// TwinCAT 3 PLC project Main
// ProgramVersion: 3.1.4023.0
// libraries:
//   Tc2_Standard, * (Beckhoff Automation GmbH)
//   Tc2_System, * (Beckhoff Automation GmbH)
//   Tc3_Module, * (Beckhoff Automation GmbH)
//   TcUnit, * (www.tcunit.org)
//   mobject-constants-datatype-limits,1.0.0,mobject
//   mobject-converters,1.0.2,mobject
// project tree:
//   / PlcTask.TcTTO
//   POUs/ MAIN.TcPOU
//   Tests/ BOOL_TO_TestSuite.TcPOU, BYTE_TO_TestSuite.TcPOU, DATE_TO_TestSuite.TcPOU, DINT_TO_TestSuite.TcPOU, DT_TO_TestSuite.TcPOU, DWORD_TO_TestSuite.TcPOU, INT_TO_TestSuite.TcPOU, LINT_TO_TestSuite.TcPOU, LREAL_TO_TestSuite.TcPOU, LWORD_TO_TestSuite.TcPOU, REAL_TO_TestSuite.TcPOU, SINT_TO_TestSuite.TcPOU, STRING_TO_TestSuite.TcPOU, TIME_TO_TestSuite.TcPOU, TOD_TO_TestSuite.TcPOU, UDINT_TO_TestSuite.TcPOU, UINT_TO_TestSuite.TcPOU, ULINT_TO_TestSuite.TcPOU, USINT_TO_TestSuite.TcPOU, WORD_TO_TestSuite.TcPOU
// real-time tasks:
//   TASK PlcTask: cycle T#10ms, priority 20, ADS port 350

CONFIGURATION Main
    RESOURCE PLC ON TwinCAT3
        TASK PlcTask(INTERVAL := T#10ms, PRIORITY := 20);
        PROGRAM MAIN WITH PlcTask : MAIN;
    END_RESOURCE
END_CONFIGURATION

// ---- POUs/MAIN.TcPOU
PROGRAM MAIN
VAR
	BOOL_TO_TestSuite : BOOL_TO_TestSuite;
	BYTE_TO_TestSuite : BYTE_TO_TestSuite;
	WORD_TO_TestSuite : WORD_TO_TestSuite;
	DWORD_TO_TestSuite : DWORD_TO_TestSuite;
	LWORD_TO_TestSuite : LWORD_TO_TestSuite;
	SINT_TO_TestSuite : SINT_TO_TestSuite;
	INT_TO_TestSuite : INT_TO_TestSuite;
	DINT_TO_TestSuite : DINT_TO_TestSuite;
	LINT_TO_TestSuite : LINT_TO_TestSuite;
	USINT_TO_TestSuite : USINT_TO_TestSuite;
	UINT_TO_TestSuite : UINT_TO_TestSuite;
	UDINT_TO_TestSuite : UDINT_TO_TestSuite;
	ULINT_TO_TestSuite : ULINT_TO_TestSuite;
	REAL_TO_TestSuite : REAL_TO_TestSuite;
	LREAL_TO_TestSuite : LREAL_TO_TestSuite;
	TIME_TO_TestSuite : TIME_TO_TestSuite;
	TOD_TO_TestSuite : TOD_TO_TestSuite;
	DATE_TO_TestSuite : DATE_TO_TestSuite;
	DT_TO_TestSuite : DT_TO_TestSuite;
	STRING_TO_TestSuite : STRING_TO_TestSuite;
END_VAR

TcUnit.RUN();

END_PROGRAM

// ---- Tests/BOOL_TO_TestSuite.TcPOU
FUNCTION_BLOCK PUBLIC BOOL_TO_TestSuite EXTENDS TcUnit.FB_TestSuite
VAR
END_VAR

Check_BOOL_TO_BOOL_Max();
Check_BOOL_TO_BOOL_Min();
Check_BOOL_TO_BYTE_Max();
Check_BOOL_TO_BYTE_Min();
Check_BOOL_TO_WORD_Max();
Check_BOOL_TO_WORD_Min();
Check_BOOL_TO_DWORD_Max();
Check_BOOL_TO_DWORD_Min();
Check_BOOL_TO_LWORD_Max();
Check_BOOL_TO_LWORD_Min();
Check_BOOL_TO_SINT_Max();
Check_BOOL_TO_SINT_Min();
Check_BOOL_TO_INT_Max();
Check_BOOL_TO_INT_Min();
Check_BOOL_TO_DINT_Max();
Check_BOOL_TO_DINT_Min();
Check_BOOL_TO_LINT_Max();
Check_BOOL_TO_LINT_Min();
Check_BOOL_TO_USINT_Max();
Check_BOOL_TO_USINT_Min();
Check_BOOL_TO_UINT_Max();
Check_BOOL_TO_UINT_Min();
Check_BOOL_TO_UDINT_Max();
Check_BOOL_TO_UDINT_Min();
Check_BOOL_TO_ULINT_Max();
Check_BOOL_TO_ULINT_Min();
Check_BOOL_TO_REAL_Max();
Check_BOOL_TO_REAL_Min();
Check_BOOL_TO_LREAL_Max();
Check_BOOL_TO_LREAL_Min();
Check_BOOL_TO_TIME_Max();
Check_BOOL_TO_TIME_Min();
Check_BOOL_TO_TOD_Max();
Check_BOOL_TO_TOD_Min();
Check_BOOL_TO_DATE_Max();
Check_BOOL_TO_DATE_Min();
Check_BOOL_TO_DT_Max();
Check_BOOL_TO_DT_Min();
Check_BOOL_TO_STRING_Max();
Check_BOOL_TO_STRING_Min();

METHOD PUBLIC Check_BOOL_TO_BOOL_Min
VAR
	value : BOOL := DatatypeLimits.BOOL_MIN_VALUE;
	actual : BOOL;
	converted : BOOL;
	equal : BOOL;
END_VAR
TEST('Check_BOOL_TO_BOOL_Min');

// @TEST-RUN
converted := TryConvert_BOOL_TO_Destination(value, actual);
equal := actual = value;

// @TEST-ASSERT
AssertTrue(Condition := equal, Message := 'Did not convert BOOL to BOOL correctly');
AssertTrue(Condition := converted, Message := 'Did not report BOOL to BOOL conversion was successful');

TEST_FINISHED();
END_METHOD

METHOD PUBLIC Check_BOOL_TO_BOOL_Max
VAR
	value : BOOL := DatatypeLimits.BOOL_MAX_VALUE;
	actual : BOOL;
	converted : BOOL;
	equal : BOOL;
END_VAR
TEST('Check_BOOL_TO_BOOL_Max');

// @TEST-RUN
converted := TryConvert_BOOL_TO_Destination(value, actual);
equal := actual = value;

// @TEST-ASSERT
AssertTrue(Condition := equal, Message := 'Did not convert BOOL to BOOL correctly');
AssertTrue(Condition := converted, Message := 'Did not report BOOL to BOOL conversion was successful');

TEST_FINISHED();
END_METHOD

METHOD PUBLIC Check_BOOL_TO_BYTE_Min
VAR
	value : BOOL := DatatypeLimits.BOOL_MIN_VALUE;
	actual : BYTE;
	converted : BOOL;
	equal : BOOL;
END_VAR
TEST('Check_BOOL_TO_BYTE_Min');

// @TEST-RUN
converted := TryConvert_BOOL_TO_Destination(value, actual);
equal := actual = BOOL_TO_BYTE(value);

// @TEST-ASSERT
AssertTrue(Condition := equal, Message := 'Did not convert BOOL to BYTE correctly');
AssertTrue(Condition := converted, Message := 'Did not report BOOL to BYTE conversion was successful');

TEST_FINISHED();
END_METHOD

METHOD PUBLIC Check_BOOL_TO_BYTE_Max
VAR
	value : BOOL := DatatypeLimits.BOOL_MAX_VALUE;
	actual : BYTE;
	converted : BOOL;
	equal : BOOL;
END_VAR
TEST('Check_BOOL_TO_BYTE_Max');

// @TEST-RUN
converted := TryConvert_BOOL_TO_Destination(value, actual);
equal := actual = BOOL_TO_BYTE(value);

// @TEST-ASSERT
AssertTrue(Condition := equal, Message := 'Did not convert BOOL to BYTE correctly');
AssertTrue(Condition := converted, Message := 'Did not report BOOL to BYTE conversion was successful');

TEST_FINISHED();
END_METHOD

METHOD PUBLIC Check_BOOL_TO_DATE_Min
VAR
	value : BOOL := DatatypeLimits.BOOL_MIN_VALUE;
	actual : DATE;
	converted : BOOL;
	equal : BOOL;
END_VAR
TEST('Check_BOOL_TO_DATE_Min');

// @TEST-RUN
converted := TryConvert_BOOL_TO_Destination(value, actual);
equal := actual = BOOL_TO_DATE(value);

// @TEST-ASSERT
AssertTrue(Condition := equal, Message := 'Did not convert BOOL to DATE correctly');
AssertTrue(Condition := converted, Message := 'Did not report BOOL to DATE conversion was successful');

TEST_FINISHED();
END_METHOD

METHOD PUBLIC Check_BOOL_TO_DATE_Max
VAR
	value : BOOL := DatatypeLimits.BOOL_MAX_VALUE;
	actual : DATE;
	converted : BOOL;
	equal : BOOL;
END_VAR
TEST('Check_BOOL_TO_DATE_Max');

// @TEST-RUN
converted := TryConvert_BOOL_TO_Destination(value, actual);
equal := actual = BOOL_TO_DATE(value);

// @TEST-ASSERT
AssertTrue(Condition := equal, Message := 'Did not convert BOOL to DATE correctly');
AssertTrue(Condition := converted, Message := 'Did not report BOOL to DATE conversion was successful');

TEST_FINISHED();
END_METHOD

METHOD PUBLIC Check_BOOL_TO_DINT_Min
VAR
	value : BOOL := DatatypeLimits.BOOL_MIN_VALUE;
	actual : DINT;
	converted : BOOL;
	equal : BOOL;
END_VAR
TEST('Check_BOOL_TO_DINT_Min');

// @TEST-RUN
converted := TryConvert_BOOL_TO_Destination(value, actual);
equal := actual = BOOL_TO_DINT(value);

// @TEST-ASSERT
AssertTrue(Condition := equal, Message := 'Did not convert BOOL to DINT correctly');
AssertTrue(Condition := converted, Message := 'Did not report BOOL to DINT conversion was successful');

TEST_FINISHED();
END_METHOD

METHOD PUBLIC Check_BOOL_TO_DINT_Max
VAR
	value : BOOL := DatatypeLimits.BOOL_MAX_VALUE;
	actual : DINT;
	converted : BOOL;
	equal : BOOL;
END_VAR
TEST('Check_BOOL_TO_DINT_Max');

// @TEST-RUN
converted := TryConvert_BOOL_TO_Destination(value, actual);
equal := actual = BOOL_TO_DINT(value);

// @TEST-ASSERT
AssertTrue(Condition := equal, Message := 'Did not convert BOOL to DINT correctly');
AssertTrue(Condition := converted, Message := 'Did not report BOOL to DINT conversion was successful');

TEST_FINISHED();
END_METHOD

METHOD PUBLIC Check_BOOL_TO_DT_Min
VAR
	value : BOOL := DatatypeLimits.BOOL_MIN_VALUE;
	actual : DT;
	converted : BOOL;
	equal : BOOL;
END_VAR
TEST('Check_BOOL_TO_DT_Min');

// @TEST-RUN
converted := TryConvert_BOOL_TO_Destination(value, actual);
equal := actual = BOOL_TO_DT(value);

// @TEST-ASSERT
AssertTrue(Condition := equal, Message := 'Did not convert BOOL to DT correctly');
AssertTrue(Condition := converted, Message := 'Did not report BOOL to DT conversion was successful');

TEST_FINISHED();
END_METHOD

METHOD PUBLIC Check_BOOL_TO_DT_Max
VAR
	value : BOOL := DatatypeLimits.BOOL_MAX_VALUE;
	actual : DT;
	converted : BOOL;
	equal : BOOL;
END_VAR
TEST('Check_BOOL_TO_DT_Max');

// @TEST-RUN
converted := TryConvert_BOOL_TO_Destination(value, actual);
equal := actual = BOOL_TO_DT(value);

// @TEST-ASSERT
AssertTrue(Condition := equal, Message := 'Did not convert BOOL to DT correctly');
AssertTrue(Condition := converted, Message := 'Did not report BOOL to DT conversion was successful');

TEST_FINISHED();
END_METHOD

METHOD PUBLIC Check_BOOL_TO_DWORD_Min
VAR
	value : BOOL := DatatypeLimits.BOOL_MIN_VALUE;
	actual : DWORD;
	converted : BOOL;
	equal : BOOL;
END_VAR
TEST('Check_BOOL_TO_DWORD_Min');

// @TEST-RUN
converted := TryConvert_BOOL_TO_Destination(value, actual);
equal := actual = BOOL_TO_DWORD(value);

// @TEST-ASSERT
AssertTrue(Condition := equal, Message := 'Did not convert BOOL to DWORD correctly');
AssertTrue(Condition := converted, Message := 'Did not report BOOL to DWORD conversion was successful');

TEST_FINISHED();
END_METHOD

METHOD PUBLIC Check_BOOL_TO_DWORD_Max
VAR
	value : BOOL := DatatypeLimits.BOOL_MAX_VALUE;
	actual : DWORD;
	converted : BOOL;
	equal : BOOL;
END_VAR
TEST('Check_BOOL_TO_DWORD_Max');

// @TEST-RUN
converted := TryConvert_BOOL_TO_Destination(value, actual);
equal := actual = BOOL_TO_DWORD(value);

// @TEST-ASSERT
AssertTrue(Condition := equal, Message := 'Did not convert BOOL to DWORD correctly');
AssertTrue(Condition := converted, Message := 'Did not report BOOL to DWORD conversion was successful');

TEST_FINISHED();
END_METHOD

METHOD PUBLIC Check_BOOL_TO_INT_Min
VAR
	value : BOOL := DatatypeLimits.BOOL_MIN_VALUE;
	actual : INT;
	converted : BOOL;
	equal : BOOL;
END_VAR
TEST('Check_BOOL_TO_INT_Min');

// @TEST-RUN
converted := TryConvert_BOOL_TO_Destination(value, actual);
equal := actual = BOOL_TO_INT(value);

// @TEST-ASSERT
AssertTrue(Condition := equal, Message := 'Did not convert BOOL to INT correctly');
AssertTrue(Condition := converted, Message := 'Did not report BOOL to INT conversion was successful');

TEST_FINISHED();
END_METHOD

METHOD PUBLIC Check_BOOL_TO_INT_Max
VAR
	value : BOOL := DatatypeLimits.BOOL_MAX_VALUE;
	actual : INT;
	converted : BOOL;
	equal : BOOL;
END_VAR
TEST('Check_BOOL_TO_INT_Max');

// @TEST-RUN
converted := TryConvert_BOOL_TO_Destination(value, actual);
equal := actual = BOOL_TO_INT(value);

// @TEST-ASSERT
AssertTrue(Condition := equal, Message := 'Did not convert BOOL to INT correctly');
AssertTrue(Condition := converted, Message := 'Did not report BOOL to INT conversion was successful');

TEST_FINISHED();
END_METHOD

METHOD PUBLIC Check_BOOL_TO_LINT_Min
VAR
	value : BOOL := DatatypeLimits.BOOL_MIN_VALUE;
	actual : LINT;
	converted : BOOL;
	equal : BOOL;
END_VAR
TEST('Check_BOOL_TO_LINT_Min');

// @TEST-RUN
converted := TryConvert_BOOL_TO_Destination(value, actual);
equal := actual = BOOL_TO_LINT(value);

// @TEST-ASSERT
AssertTrue(Condition := equal, Message := 'Did not convert BOOL to LINT correctly');
AssertTrue(Condition := converted, Message := 'Did not report BOOL to LINT conversion was successful');

TEST_FINISHED();
END_METHOD

METHOD PUBLIC Check_BOOL_TO_LINT_Max
VAR
	value : BOOL := DatatypeLimits.BOOL_MAX_VALUE;
	actual : LINT;
	converted : BOOL;
	equal : BOOL;
END_VAR
TEST('Check_BOOL_TO_LINT_Max');

// @TEST-RUN
converted := TryConvert_BOOL_TO_Destination(value, actual);
equal := actual = BOOL_TO_LINT(value);

// @TEST-ASSERT
AssertTrue(Condition := equal, Message := 'Did not convert BOOL to LINT correctly');
AssertTrue(Condition := converted, Message := 'Did not report BOOL to LINT conversion was successful');

TEST_FINISHED();
END_METHOD

METHOD PUBLIC Check_BOOL_TO_LREAL_Min
VAR
	value : BOOL := DatatypeLimits.BOOL_MIN_VALUE;
	actual : LREAL;
	converted : BOOL;
	equal : BOOL;
END_VAR
TEST('Check_BOOL_TO_LREAL_Min');

// @TEST-RUN
converted := TryConvert_BOOL_TO_Destination(value, actual);
equal := actual = BOOL_TO_LREAL(value);

// @TEST-ASSERT
AssertTrue(Condition := equal, Message := 'Did not convert BOOL to LREAL correctly');
AssertTrue(Condition := converted, Message := 'Did not report BOOL to LREAL conversion was successful');

TEST_FINISHED();
END_METHOD

METHOD PUBLIC Check_BOOL_TO_LREAL_Max
VAR
	value : BOOL := DatatypeLimits.BOOL_MAX_VALUE;
	actual : LREAL;
	converted : BOOL;
	equal : BOOL;
END_VAR
TEST('Check_BOOL_TO_LREAL_Max');

// @TEST-RUN
converted := TryConvert_BOOL_TO_Destination(value, actual);
equal := actual = BOOL_TO_LREAL(value);

// @TEST-ASSERT
AssertTrue(Condition := equal, Message := 'Did not convert BOOL to LREAL correctly');
AssertTrue(Condition := converted, Message := 'Did not report BOOL to LREAL conversion was successful');

TEST_FINISHED();
END_METHOD

METHOD PUBLIC Check_BOOL_TO_LWORD_Min
VAR
	value : BOOL := DatatypeLimits.BOOL_MIN_VALUE;
	actual : LWORD;
	converted : BOOL;
	equal : BOOL;
END_VAR
TEST('Check_BOOL_TO_LWORD_Min');

// @TEST-RUN
converted := TryConvert_BOOL_TO_Destination(value, actual);
equal := actual = BOOL_TO_LWORD(value);

// @TEST-ASSERT
AssertTrue(Condition := equal, Message := 'Did not convert BOOL to LWORD correctly');
AssertTrue(Condition := converted, Message := 'Did not report BOOL to LWORD conversion was successful');

TEST_FINISHED();
END_METHOD

METHOD PUBLIC Check_BOOL_TO_LWORD_Max
VAR
	value : BOOL := DatatypeLimits.BOOL_MAX_VALUE;
	actual : LWORD;
	converted : BOOL;
	equal : BOOL;
END_VAR
TEST('Check_BOOL_TO_LWORD_Max');

// @TEST-RUN
converted := TryConvert_BOOL_TO_Destination(value, actual);
equal := actual = BOOL_TO_LWORD(value);

// @TEST-ASSERT
AssertTrue(Condition := equal, Message := 'Did not convert BOOL to LWORD correctly');
AssertTrue(Condition := converted, Message := 'Did not report BOOL to LWORD conversion was successful');

TEST_FINISHED();
END_METHOD

METHOD PUBLIC Check_BOOL_TO_REAL_Min
VAR
	value : BOOL := DatatypeLimits.BOOL_MIN_VALUE;
	actual : REAL;
	converted : BOOL;
	equal : BOOL;
END_VAR
TEST('Check_BOOL_TO_REAL_Min');

// @TEST-RUN
converted := TryConvert_BOOL_TO_Destination(value, actual);
equal := actual = BOOL_TO_REAL(value);

// @TEST-ASSERT
AssertTrue(Condition := equal, Message := 'Did not convert BOOL to REAL correctly');
AssertTrue(Condition := converted, Message := 'Did not report BOOL to REAL conversion was successful');

TEST_FINISHED();
END_METHOD

METHOD PUBLIC Check_BOOL_TO_REAL_Max
VAR
	value : BOOL := DatatypeLimits.BOOL_MAX_VALUE;
	actual : REAL;
	converted : BOOL;
	equal : BOOL;
END_VAR
TEST('Check_BOOL_TO_REAL_Max');

// @TEST-RUN
converted := TryConvert_BOOL_TO_Destination(value, actual);
equal := actual = BOOL_TO_REAL(value);

// @TEST-ASSERT
AssertTrue(Condition := equal, Message := 'Did not convert BOOL to REAL correctly');
AssertTrue(Condition := converted, Message := 'Did not report BOOL to REAL conversion was successful');

TEST_FINISHED();
END_METHOD

METHOD PUBLIC Check_BOOL_TO_SINT_Min
VAR
	value : BOOL := DatatypeLimits.BOOL_MIN_VALUE;
	actual : SINT;
	converted : BOOL;
	equal : BOOL;
END_VAR
TEST('Check_BOOL_TO_SINT_Min');

// @TEST-RUN
converted := TryConvert_BOOL_TO_Destination(value, actual);
equal := actual = BOOL_TO_SINT(value);

// @TEST-ASSERT
AssertTrue(Condition := equal, Message := 'Did not convert BOOL to SINT correctly');
AssertTrue(Condition := converted, Message := 'Did not report BOOL to SINT conversion was successful');

TEST_FINISHED();
END_METHOD

METHOD PUBLIC Check_BOOL_TO_SINT_Max
VAR
	value : BOOL := DatatypeLimits.BOOL_MAX_VALUE;
	actual : SINT;
	converted : BOOL;
	equal : BOOL;
END_VAR
TEST('Check_BOOL_TO_SINT_Max');

// @TEST-RUN
converted := TryConvert_BOOL_TO_Destination(value, actual);
equal := actual = BOOL_TO_SINT(value);

// @TEST-ASSERT
AssertTrue(Condition := equal, Message := 'Did not convert BOOL to SINT correctly');
AssertTrue(Condition := converted, Message := 'Did not report BOOL to SINT conversion was successful');

TEST_FINISHED();
END_METHOD

METHOD PUBLIC Check_BOOL_TO_STRING_Min
VAR
	value : BOOL := DatatypeLimits.BOOL_MIN_VALUE;
	actual : STRING;
	converted : BOOL;
	equal : BOOL;
END_VAR
TEST('Check_BOOL_TO_STRING_Min');

// @TEST-RUN
converted := TryConvert_BOOL_TO_Destination(value, actual);
equal := actual = BOOL_TO_STRING(value);

// @TEST-ASSERT
AssertTrue(Condition := equal, Message := 'Did not convert BOOL to STRING correctly');
AssertTrue(Condition := converted, Message := 'Did not report BOOL to STRING conversion was successful');

TEST_FINISHED();
END_METHOD

METHOD PUBLIC Check_BOOL_TO_STRING_Max
VAR
	value : BOOL := DatatypeLimits.BOOL_MAX_VALUE;
	actual : STRING;
	converted : BOOL;
	equal : BOOL;
END_VAR
TEST('Check_BOOL_TO_STRING_Max');

// @TEST-RUN
converted := TryConvert_BOOL_TO_Destination(value, actual);
equal := actual = BOOL_TO_STRING(value);

// @TEST-ASSERT
AssertTrue(Condition := equal, Message := 'Did not convert BOOL to STRING correctly');
AssertTrue(Condition := converted, Message := 'Did not report BOOL to STRING conversion was successful');

TEST_FINISHED();
END_METHOD

METHOD PUBLIC Check_BOOL_TO_TIME_Min
VAR
	value : BOOL := DatatypeLimits.BOOL_MIN_VALUE;
	actual : TIME;
	converted : BOOL;
	equal : BOOL;
END_VAR
TEST('Check_BOOL_TO_TIME_Min');

// @TEST-RUN
converted := TryConvert_BOOL_TO_Destination(value, actual);
equal := actual = BOOL_TO_TIME(value);

// @TEST-ASSERT
AssertTrue(Condition := equal, Message := 'Did not convert BOOL to TIME correctly');
AssertTrue(Condition := converted, Message := 'Did not report BOOL to TIME conversion was successful');

TEST_FINISHED();
END_METHOD

METHOD PUBLIC Check_BOOL_TO_TIME_Max
VAR
	value : BOOL := DatatypeLimits.BOOL_MAX_VALUE;
	actual : TIME;
	converted : BOOL;
	equal : BOOL;
END_VAR
TEST('Check_BOOL_TO_TIME_Max');

// @TEST-RUN
converted := TryConvert_BOOL_TO_Destination(value, actual);
equal := actual = BOOL_TO_TIME(value);

// @TEST-ASSERT
AssertTrue(Condition := equal, Message := 'Did not convert BOOL to TIME correctly');
AssertTrue(Condition := converted, Message := 'Did not report BOOL to TIME conversion was successful');

TEST_FINISHED();
END_METHOD

METHOD PUBLIC Check_BOOL_TO_TOD_Min
VAR
	value : BOOL := DatatypeLimits.BOOL_MIN_VALUE;
	actual : TOD;
	converted : BOOL;
	equal : BOOL;
END_VAR
TEST('Check_BOOL_TO_TOD_Min');

// @TEST-RUN
converted := TryConvert_BOOL_TO_Destination(value, actual);
equal := actual = BOOL_TO_TOD(value);

// @TEST-ASSERT
AssertTrue(Condition := equal, Message := 'Did not convert BOOL to TOD correctly');
AssertTrue(Condition := converted, Message := 'Did not report BOOL to TOD conversion was successful');

TEST_FINISHED();
END_METHOD

METHOD PUBLIC Check_BOOL_TO_TOD_Max
VAR
	value : BOOL := DatatypeLimits.BOOL_MAX_VALUE;
	actual : TOD;
	converted : BOOL;
	equal : BOOL;
END_VAR
TEST('Check_BOOL_TO_TOD_Max');

// @TEST-RUN
converted := TryConvert_BOOL_TO_Destination(value, actual);
equal := actual = BOOL_TO_TOD(value);

// @TEST-ASSERT
AssertTrue(Condition := equal, Message := 'Did not convert BOOL to TOD correctly');
AssertTrue(Condition := converted, Message := 'Did not report BOOL to TOD conversion was successful');

TEST_FINISHED();
END_METHOD

METHOD PUBLIC Check_BOOL_TO_UDINT_Min
VAR
	value : BOOL := DatatypeLimits.BOOL_MIN_VALUE;
	actual : UDINT;
	converted : BOOL;
	equal : BOOL;
END_VAR
TEST('Check_BOOL_TO_UDINT_Min');

// @TEST-RUN
converted := TryConvert_BOOL_TO_Destination(value, actual);
equal := actual = BOOL_TO_UDINT(value);

// @TEST-ASSERT
AssertTrue(Condition := equal, Message := 'Did not convert BOOL to UDINT correctly');
AssertTrue(Condition := converted, Message := 'Did not report BOOL to UDINT conversion was successful');

TEST_FINISHED();
END_METHOD

METHOD PUBLIC Check_BOOL_TO_UDINT_Max
VAR
	value : BOOL := DatatypeLimits.BOOL_MAX_VALUE;
	actual : UDINT;
	converted : BOOL;
	equal : BOOL;
END_VAR
TEST('Check_BOOL_TO_UDINT_Max');

// @TEST-RUN
converted := TryConvert_BOOL_TO_Destination(value, actual);
equal := actual = BOOL_TO_UDINT(value);

// @TEST-ASSERT
AssertTrue(Condition := equal, Message := 'Did not convert BOOL to UDINT correctly');
AssertTrue(Condition := converted, Message := 'Did not report BOOL to UDINT conversion was successful');

TEST_FINISHED();
END_METHOD

METHOD PUBLIC Check_BOOL_TO_UINT_Min
VAR
	value : BOOL := DatatypeLimits.BOOL_MIN_VALUE;
	actual : UINT;
	converted : BOOL;
	equal : BOOL;
END_VAR
TEST('Check_BOOL_TO_UINT_Min');

// @TEST-RUN
converted := TryConvert_BOOL_TO_Destination(value, actual);
equal := actual = BOOL_TO_UINT(value);

// @TEST-ASSERT
AssertTrue(Condition := equal, Message := 'Did not convert BOOL to UINT correctly');
AssertTrue(Condition := converted, Message := 'Did not report BOOL to UINT conversion was successful');

TEST_FINISHED();
END_METHOD

METHOD PUBLIC Check_BOOL_TO_UINT_Max
VAR
	value : BOOL := DatatypeLimits.BOOL_MAX_VALUE;
	actual : UINT;
	converted : BOOL;
	equal : BOOL;
END_VAR
TEST('Check_BOOL_TO_UINT_Max');

// @TEST-RUN
converted := TryConvert_BOOL_TO_Destination(value, actual);
equal := actual = BOOL_TO_UINT(value);

// @TEST-ASSERT
AssertTrue(Condition := equal, Message := 'Did not convert BOOL to UINT correctly');
AssertTrue(Condition := converted, Message := 'Did not report BOOL to UINT conversion was successful');

TEST_FINISHED();
END_METHOD

METHOD PUBLIC Check_BOOL_TO_ULINT_Min
VAR
	value : BOOL := DatatypeLimits.BOOL_MIN_VALUE;
	actual : ULINT;
	converted : BOOL;
	equal : BOOL;
END_VAR
TEST('Check_BOOL_TO_ULINT_Min');

// @TEST-RUN
converted := TryConvert_BOOL_TO_Destination(value, actual);
equal := actual = BOOL_TO_ULINT(value);

// @TEST-ASSERT
AssertTrue(Condition := equal, Message := 'Did not convert BOOL to ULINT correctly');
AssertTrue(Condition := converted, Message := 'Did not report BOOL to ULINT conversion was successful');

TEST_FINISHED();
END_METHOD

METHOD PUBLIC Check_BOOL_TO_ULINT_Max
VAR
	value : BOOL := DatatypeLimits.BOOL_MAX_VALUE;
	actual : ULINT;
	converted : BOOL;
	equal : BOOL;
END_VAR
TEST('Check_BOOL_TO_ULINT_Max');

// @TEST-RUN
converted := TryConvert_BOOL_TO_Destination(value, actual);
equal := actual = BOOL_TO_ULINT(value);

// @TEST-ASSERT
AssertTrue(Condition := equal, Message := 'Did not convert BOOL to ULINT correctly');
AssertTrue(Condition := converted, Message := 'Did not report BOOL to ULINT conversion was successful');

TEST_FINISHED();
END_METHOD

METHOD PUBLIC Check_BOOL_TO_USINT_Min
VAR
	value : BOOL := DatatypeLimits.BOOL_MIN_VALUE;
	actual : USINT;
	converted : BOOL;
	equal : BOOL;
END_VAR
TEST('Check_BOOL_TO_USINT_Min');

// @TEST-RUN
converted := TryConvert_BOOL_TO_Destination(value, actual);
equal := actual = BOOL_TO_USINT(value);

// @TEST-ASSERT
AssertTrue(Condition := equal, Message := 'Did not convert BOOL to USINT correctly');
AssertTrue(Condition := converted, Message := 'Did not report BOOL to USINT conversion was successful');

TEST_FINISHED();
END_METHOD

METHOD PUBLIC Check_BOOL_TO_USINT_Max
VAR
	value : BOOL := DatatypeLimits.BOOL_MAX_VALUE;
	actual : USINT;
	converted : BOOL;
	equal : BOOL;
END_VAR
TEST('Check_BOOL_TO_USINT_Max');

// @TEST-RUN
converted := TryConvert_BOOL_TO_Destination(value, actual);
equal := actual = BOOL_TO_USINT(value);

// @TEST-ASSERT
AssertTrue(Condition := equal, Message := 'Did not convert BOOL to USINT correctly');
AssertTrue(Condition := converted, Message := 'Did not report BOOL to USINT conversion was successful');

TEST_FINISHED();
END_METHOD

METHOD PUBLIC Check_BOOL_TO_WORD_Min
VAR
	value : BOOL := DatatypeLimits.BOOL_MIN_VALUE;
	actual : WORD;
	converted : BOOL;
	equal : BOOL;
END_VAR
TEST('Check_BOOL_TO_WORD_Min');

// @TEST-RUN
converted := TryConvert_BOOL_TO_Destination(value, actual);
equal := actual = BOOL_TO_WORD(value);

// @TEST-ASSERT
AssertTrue(Condition := equal, Message := 'Did not convert BOOL to WORD correctly');
AssertTrue(Condition := converted, Message := 'Did not report BOOL to WORD conversion was successful');

TEST_FINISHED();
END_METHOD

METHOD PUBLIC Check_BOOL_TO_WORD_Max
VAR
	value : BOOL := DatatypeLimits.BOOL_MAX_VALUE;
	actual : WORD;
	converted : BOOL;
	equal : BOOL;
END_VAR
TEST('Check_BOOL_TO_WORD_Max');

// @TEST-RUN
converted := TryConvert_BOOL_TO_Destination(value, actual);
equal := actual = BOOL_TO_WORD(value);

// @TEST-ASSERT
AssertTrue(Condition := equal, Message := 'Did not convert BOOL to WORD correctly');
AssertTrue(Condition := converted, Message := 'Did not report BOOL to WORD conversion was successful');

TEST_FINISHED();
END_METHOD

END_FUNCTION_BLOCK

// ---- Tests/BYTE_TO_TestSuite.TcPOU
FUNCTION_BLOCK PUBLIC BYTE_TO_TestSuite EXTENDS TcUnit.FB_TestSuite
VAR
END_VAR

Check_BYTE_TO_BOOL_Max();
Check_BYTE_TO_BOOL_Min();
Check_BYTE_TO_BYTE_Max();
Check_BYTE_TO_BYTE_Min();
Check_BYTE_TO_WORD_Max();
Check_BYTE_TO_WORD_Min();
Check_BYTE_TO_DWORD_Max();
Check_BYTE_TO_DWORD_Min();
Check_BYTE_TO_LWORD_Max();
Check_BYTE_TO_LWORD_Min();
Check_BYTE_TO_SINT_Max();
Check_BYTE_TO_SINT_Min();
Check_BYTE_TO_SINT_TooHigh();
Check_BYTE_TO_INT_Max();
Check_BYTE_TO_INT_Min();
Check_BYTE_TO_DINT_Max();
Check_BYTE_TO_DINT_Min();
Check_BYTE_TO_LINT_Max();
Check_BYTE_TO_LINT_Min();
Check_BYTE_TO_USINT_Max();
Check_BYTE_TO_USINT_Min();
Check_BYTE_TO_UINT_Max();
Check_BYTE_TO_UINT_Min();
Check_BYTE_TO_UDINT_Max();
Check_BYTE_TO_UDINT_Min();
Check_BYTE_TO_ULINT_Max();
Check_BYTE_TO_ULINT_Min();
Check_BYTE_TO_REAL_Max();
Check_BYTE_TO_REAL_Min();
Check_BYTE_TO_LREAL_Max();
Check_BYTE_TO_LREAL_Min();
Check_BYTE_TO_TIME_Max();
Check_BYTE_TO_TIME_Min();
Check_BYTE_TO_TOD_Max();
Check_BYTE_TO_TOD_Min();
Check_BYTE_TO_DATE_Max();
Check_BYTE_TO_DATE_Min();
Check_BYTE_TO_DT_Max();
Check_BYTE_TO_DT_Min();
Check_BYTE_TO_STRING_Max();
Check_BYTE_TO_STRING_Min();

METHOD PUBLIC Check_BYTE_TO_BOOL_Min
VAR
	value : BYTE := DatatypeLimits.BYTE_MIN_VALUE;
	actual : BOOL;
	converted : BOOL;
	equal : BOOL;
END_VAR
TEST('Check_BYTE_TO_BOOL_Min');

// @TEST-RUN
converted := TryConvert_BYTE_TO_Destination(value, actual);
equal := actual = BYTE_TO_BOOL(value);

// @TEST-ASSERT
AssertTrue(Condition := equal, Message := 'Did not convert BYTE to BOOL correctly');
AssertTrue(Condition := converted, Message := 'Did not report BYTE to BOOL conversion was successful');

TEST_FINISHED();
END_METHOD

METHOD PUBLIC Check_BYTE_TO_BOOL_Max
VAR
	value : BYTE := DatatypeLimits.BYTE_MAX_VALUE;
	actual : BOOL;
	converted : BOOL;
	equal : BOOL;
END_VAR
TEST('Check_BYTE_TO_BOOL_Max');

// @TEST-RUN
converted := TryConvert_BYTE_TO_Destination(value, actual);
equal := actual = BYTE_TO_BOOL(value);

// @TEST-ASSERT
AssertTrue(Condition := equal, Message := 'Did not convert BYTE to BOOL correctly');
AssertTrue(Condition := converted, Message := 'Did not report BYTE to BOOL conversion was successful');

TEST_FINISHED();
END_METHOD

METHOD PUBLIC Check_BYTE_TO_BYTE_Min
VAR
	value : BYTE := DatatypeLimits.BYTE_MIN_VALUE;
	actual : BYTE;
	converted : BOOL;
	equal : BOOL;
END_VAR
TEST('Check_BYTE_TO_BYTE_Min');

// @TEST-RUN
converted := TryConvert_BYTE_TO_Destination(value, actual);
equal := actual = value;

// @TEST-ASSERT
AssertTrue(Condition := equal, Message := 'Did not convert BYTE to BYTE correctly');
AssertTrue(Condition := converted, Message := 'Did not report BYTE to BYTE conversion was successful');

TEST_FINISHED();
END_METHOD

METHOD PUBLIC Check_BYTE_TO_BYTE_Max
VAR
	value : BYTE := DatatypeLimits.BYTE_MAX_VALUE;
	actual : BYTE;
	converted : BOOL;
	equal : BOOL;
END_VAR
TEST('Check_BYTE_TO_BYTE_Max');

// @TEST-RUN
converted := TryConvert_BYTE_TO_Destination(value, actual);
equal := actual = value;

// @TEST-ASSERT
AssertTrue(Condition := equal, Message := 'Did not convert BYTE to BYTE correctly');
AssertTrue(Condition := converted, Message := 'Did not report BYTE to BYTE conversion was successful');

TEST_FINISHED();
END_METHOD

METHOD PUBLIC Check_BYTE_TO_DATE_Min
VAR
	value : BYTE := DatatypeLimits.BYTE_MIN_VALUE;
	actual : DATE;
	converted : BOOL;
	equal : BOOL;
END_VAR
TEST('Check_BYTE_TO_DATE_Min');

// @TEST-RUN
converted := TryConvert_BYTE_TO_Destination(value, actual);
equal := actual = BYTE_TO_DATE(value);

// @TEST-ASSERT
AssertTrue(Condition := equal, Message := 'Did not convert BYTE to DATE correctly');
AssertTrue(Condition := converted, Message := 'Did not report BYTE to DATE conversion was successful');

TEST_FINISHED();
END_METHOD

METHOD PUBLIC Check_BYTE_TO_DATE_Max
VAR
	value : BYTE := DatatypeLimits.BYTE_MAX_VALUE;
	actual : DATE;
	converted : BOOL;
	equal : BOOL;
END_VAR
TEST('Check_BYTE_TO_DATE_Max');

// @TEST-RUN
converted := TryConvert_BYTE_TO_Destination(value, actual);
equal := actual = BYTE_TO_DATE(value);

// @TEST-ASSERT
AssertTrue(Condition := equal, Message := 'Did not convert BYTE to DATE correctly');
AssertTrue(Condition := converted, Message := 'Did not report BYTE to DATE conversion was successful');

TEST_FINISHED();
END_METHOD

METHOD PUBLIC Check_BYTE_TO_DINT_Min
VAR
	value : BYTE := DatatypeLimits.BYTE_MIN_VALUE;
	actual : DINT;
	converted : BOOL;
	equal : BOOL;
END_VAR
TEST('Check_BYTE_TO_DINT_Min');

// @TEST-RUN
converted := TryConvert_BYTE_TO_Destination(value, actual);
equal := actual = BYTE_TO_DINT(value);

// @TEST-ASSERT
AssertTrue(Condition := equal, Message := 'Did not convert BYTE to DINT correctly');
AssertTrue(Condition := converted, Message := 'Did not report BYTE to DINT conversion was successful');

TEST_FINISHED();
END_METHOD

METHOD PUBLIC Check_BYTE_TO_DINT_Max
VAR
	value : BYTE := DatatypeLimits.BYTE_MAX_VALUE;
	actual : DINT;
	converted : BOOL;
	equal : BOOL;
END_VAR
TEST('Check_BYTE_TO_DINT_Max');

// @TEST-RUN
converted := TryConvert_BYTE_TO_Destination(value, actual);
equal := actual = BYTE_TO_DINT(value);

// @TEST-ASSERT
AssertTrue(Condition := equal, Message := 'Did not convert BYTE to DINT correctly');
AssertTrue(Condition := converted, Message := 'Did not report BYTE to DINT conversion was successful');

TEST_FINISHED();
END_METHOD

METHOD PUBLIC Check_BYTE_TO_DT_Min
VAR
	value : BYTE := DatatypeLimits.BYTE_MIN_VALUE;
	actual : DT;
	converted : BOOL;
	equal : BOOL;
END_VAR
TEST('Check_BYTE_TO_DT_Min');

// @TEST-RUN
converted := TryConvert_BYTE_TO_Destination(value, actual);
equal := actual = BYTE_TO_DT(value);

// @TEST-ASSERT
AssertTrue(Condition := equal, Message := 'Did not convert BYTE to DT correctly');
AssertTrue(Condition := converted, Message := 'Did not report BYTE to DT conversion was successful');

TEST_FINISHED();
END_METHOD

METHOD PUBLIC Check_BYTE_TO_DT_Max
VAR
	value : BYTE := DatatypeLimits.BYTE_MAX_VALUE;
	actual : DT;
	converted : BOOL;
	equal : BOOL;
END_VAR
TEST('Check_BYTE_TO_DT_Max');

// @TEST-RUN
converted := TryConvert_BYTE_TO_Destination(value, actual);
equal := actual = BYTE_TO_DT(value);

// @TEST-ASSERT
AssertTrue(Condition := equal, Message := 'Did not convert BYTE to DT correctly');
AssertTrue(Condition := converted, Message := 'Did not report BYTE to DT conversion was successful');

TEST_FINISHED();
END_METHOD

METHOD PUBLIC Check_BYTE_TO_DWORD_Min
VAR
	value : BYTE := DatatypeLimits.BYTE_MIN_VALUE;
	actual : DWORD;
	converted : BOOL;
	equal : BOOL;
END_VAR
TEST('Check_BYTE_TO_DWORD_Min');

// @TEST-RUN
converted := TryConvert_BYTE_TO_Destination(value, actual);
equal := actual = BYTE_TO_DWORD(value);

// @TEST-ASSERT
AssertTrue(Condition := equal, Message := 'Did not convert BYTE to DWORD correctly');
AssertTrue(Condition := converted, Message := 'Did not report BYTE to DWORD conversion was successful');

TEST_FINISHED();
END_METHOD

METHOD PUBLIC Check_BYTE_TO_DWORD_Max
VAR
	value : BYTE := DatatypeLimits.BYTE_MAX_VALUE;
	actual : DWORD;
	converted : BOOL;
	equal : BOOL;
END_VAR
TEST('Check_BYTE_TO_DWORD_Max');

// @TEST-RUN
converted := TryConvert_BYTE_TO_Destination(value, actual);
equal := actual = BYTE_TO_DWORD(value);

// @TEST-ASSERT
AssertTrue(Condition := equal, Message := 'Did not convert BYTE to DWORD correctly');
AssertTrue(Condition := converted, Message := 'Did not report BYTE to DWORD conversion was successful');

TEST_FINISHED();
END_METHOD

METHOD PUBLIC Check_BYTE_TO_INT_Min
VAR
	value : BYTE := DatatypeLimits.BYTE_MIN_VALUE;
	actual : INT;
	converted : BOOL;
	equal : BOOL;
END_VAR
TEST('Check_BYTE_TO_INT_Min');

// @TEST-RUN
converted := TryConvert_BYTE_TO_Destination(value, actual);
equal := actual = BYTE_TO_INT(value);

// @TEST-ASSERT
AssertTrue(Condition := equal, Message := 'Did not convert BYTE to INT correctly');
AssertTrue(Condition := converted, Message := 'Did not report BYTE to INT conversion was successful');

TEST_FINISHED();
END_METHOD

METHOD PUBLIC Check_BYTE_TO_INT_Max
VAR
	value : BYTE := DatatypeLimits.BYTE_MAX_VALUE;
	actual : INT;
	converted : BOOL;
	equal : BOOL;
END_VAR
TEST('Check_BYTE_TO_INT_Max');

// @TEST-RUN
converted := TryConvert_BYTE_TO_Destination(value, actual);
equal := actual = BYTE_TO_INT(value);

// @TEST-ASSERT
AssertTrue(Condition := equal, Message := 'Did not convert BYTE to INT correctly');
AssertTrue(Condition := converted, Message := 'Did not report BYTE to INT conversion was successful');

TEST_FINISHED();
END_METHOD

METHOD PUBLIC Check_BYTE_TO_LINT_Min
VAR
	value : BYTE := DatatypeLimits.BYTE_MIN_VALUE;
	actual : LINT;
	converted : BOOL;
	equal : BOOL;
END_VAR
TEST('Check_BYTE_TO_LINT_Min');

// @TEST-RUN
converted := TryConvert_BYTE_TO_Destination(value, actual);
equal := actual = BYTE_TO_LINT(value);

// @TEST-ASSERT
AssertTrue(Condition := equal, Message := 'Did not convert BYTE to LINT correctly');
AssertTrue(Condition := converted, Message := 'Did not report BYTE to LINT conversion was successful');

TEST_FINISHED();
END_METHOD

METHOD PUBLIC Check_BYTE_TO_LINT_Max
VAR
	value : BYTE := DatatypeLimits.BYTE_MAX_VALUE;
	actual : LINT;
	converted : BOOL;
	equal : BOOL;
END_VAR
TEST('Check_BYTE_TO_LINT_Max');

// @TEST-RUN
converted := TryConvert_BYTE_TO_Destination(value, actual);
equal := actual = BYTE_TO_LINT(value);

// @TEST-ASSERT
AssertTrue(Condition := equal, Message := 'Did not convert BYTE to LINT correctly');
AssertTrue(Condition := converted, Message := 'Did not report BYTE to LINT conversion was successful');

TEST_FINISHED();
END_METHOD

METHOD PUBLIC Check_BYTE_TO_LREAL_Min
VAR
	value : BYTE := DatatypeLimits.BYTE_MIN_VALUE;
	actual : LREAL;
	converted : BOOL;
	equal : BOOL;
END_VAR
TEST('Check_BYTE_TO_LREAL_Min');

// @TEST-RUN
converted := TryConvert_BYTE_TO_Destination(value, actual);
equal := actual = BYTE_TO_LREAL(value);

// @TEST-ASSERT
AssertTrue(Condition := equal, Message := 'Did not convert BYTE to LREAL correctly');
AssertTrue(Condition := converted, Message := 'Did not report BYTE to LREAL conversion was successful');

TEST_FINISHED();
END_METHOD

METHOD PUBLIC Check_BYTE_TO_LREAL_Max
VAR
	value : BYTE := DatatypeLimits.BYTE_MAX_VALUE;
	actual : LREAL;
	converted : BOOL;
	equal : BOOL;
END_VAR
TEST('Check_BYTE_TO_LREAL_Max');

// @TEST-RUN
converted := TryConvert_BYTE_TO_Destination(value, actual);
equal := actual = BYTE_TO_LREAL(value);

// @TEST-ASSERT
AssertTrue(Condition := equal, Message := 'Did not convert BYTE to LREAL correctly');
AssertTrue(Condition := converted, Message := 'Did not report BYTE to LREAL conversion was successful');

TEST_FINISHED();
END_METHOD

METHOD PUBLIC Check_BYTE_TO_LWORD_Min
VAR
	value : BYTE := DatatypeLimits.BYTE_MIN_VALUE;
	actual : LWORD;
	converted : BOOL;
	equal : BOOL;
END_VAR
TEST('Check_BYTE_TO_LWORD_Min');

// @TEST-RUN
converted := TryConvert_BYTE_TO_Destination(value, actual);
equal := actual = BYTE_TO_LWORD(value);

// @TEST-ASSERT
AssertTrue(Condition := equal, Message := 'Did not convert BYTE to LWORD correctly');
AssertTrue(Condition := converted, Message := 'Did not report BYTE to LWORD conversion was successful');

TEST_FINISHED();
END_METHOD

METHOD PUBLIC Check_BYTE_TO_LWORD_Max
VAR
	value : BYTE := DatatypeLimits.BYTE_MAX_VALUE;
	actual : LWORD;
	converted : BOOL;
	equal : BOOL;
END_VAR
TEST('Check_BYTE_TO_LWORD_Max');

// @TEST-RUN
converted := TryConvert_BYTE_TO_Destination(value, actual);
equal := actual = BYTE_TO_LWORD(value);

// @TEST-ASSERT
AssertTrue(Condition := equal, Message := 'Did not convert BYTE to LWORD correctly');
AssertTrue(Condition := converted, Message := 'Did not report BYTE to LWORD conversion was successful');

TEST_FINISHED();
END_METHOD

METHOD PUBLIC Check_BYTE_TO_REAL_Min
VAR
	value : BYTE := DatatypeLimits.BYTE_MIN_VALUE;
	actual : REAL;
	converted : BOOL;
	equal : BOOL;
END_VAR
TEST('Check_BYTE_TO_REAL_Min');

// @TEST-RUN
converted := TryConvert_BYTE_TO_Destination(value, actual);
equal := actual = BYTE_TO_REAL(value);

// @TEST-ASSERT
AssertTrue(Condition := equal, Message := 'Did not convert BYTE to REAL correctly');
AssertTrue(Condition := converted, Message := 'Did not report BYTE to REAL conversion was successful');

TEST_FINISHED();
END_METHOD

METHOD PUBLIC Check_BYTE_TO_REAL_Max
VAR
	value : BYTE := DatatypeLimits.BYTE_MAX_VALUE;
	actual : REAL;
	converted : BOOL;
	equal : BOOL;
END_VAR
TEST('Check_BYTE_TO_REAL_Max');

// @TEST-RUN
converted := TryConvert_BYTE_TO_Destination(value, actual);
equal := actual = BYTE_TO_REAL(value);

// @TEST-ASSERT
AssertTrue(Condition := equal, Message := 'Did not convert BYTE to REAL correctly');
AssertTrue(Condition := converted, Message := 'Did not report BYTE to REAL conversion was successful');

TEST_FINISHED();
END_METHOD

METHOD PUBLIC Check_BYTE_TO_SINT_Min
VAR
	value : BYTE := DatatypeLimits.BYTE_MIN_VALUE;
	actual : SINT;
	converted : BOOL;
	equal : BOOL;
END_VAR
TEST('Check_BYTE_TO_SINT_Min');

// @TEST-RUN
converted := TryConvert_BYTE_TO_Destination(value, actual);
equal := actual = BYTE_TO_SINT(value);

// @TEST-ASSERT
AssertTrue(Condition := equal, Message := 'Did not convert BYTE to SINT correctly');
AssertTrue(Condition := converted, Message := 'Did not report BYTE to SINT conversion was successful');

TEST_FINISHED();
END_METHOD

METHOD PUBLIC Check_BYTE_TO_SINT_TooHigh
VAR
	value : BYTE := DatatypeLimits.BYTE_MAX_VALUE;
	actual : SINT;
	converted : BOOL;
END_VAR
TEST('Check_BYTE_TO_SINT_TooHigh');

// @TEST-RUN
converted := TryConvert_BYTE_TO_Destination(value, actual);

// @TEST-ASSERT
AssertFalse(Condition := converted, Message := 'Did not report BYTE to SINT conversion was prevented');

TEST_FINISHED();
END_METHOD

METHOD PUBLIC Check_BYTE_TO_SINT_Max
VAR
	value : BYTE := DatatypeLimits.MAX_VALUE_OF_BYTE_WHICH_CAN_BE_HELD_IN_A_SINT;
	actual : SINT;
	converted : BOOL;
	equal : BOOL;
END_VAR
TEST('Check_BYTE_TO_SINT_Max');

// @TEST-RUN
converted := TryConvert_BYTE_TO_Destination(value, actual);
equal := actual = BYTE_TO_SINT(value);

// @TEST-ASSERT
AssertTrue(Condition := equal, Message := 'Did not convert BYTE to SINT correctly');
AssertTrue(Condition := converted, Message := 'Did not report BYTE to SINT conversion was successful');

TEST_FINISHED();
END_METHOD

METHOD PUBLIC Check_BYTE_TO_STRING_Min
VAR
	value : BYTE := DatatypeLimits.BYTE_MIN_VALUE;
	actual : STRING;
	converted : BOOL;
	equal : BOOL;
END_VAR
TEST('Check_BYTE_TO_STRING_Min');

// @TEST-RUN
converted := TryConvert_BYTE_TO_Destination(value, actual);
equal := actual = BYTE_TO_STRING(value);

// @TEST-ASSERT
AssertTrue(Condition := equal, Message := 'Did not convert BYTE to STRING correctly');
AssertTrue(Condition := converted, Message := 'Did not report BYTE to STRING conversion was successful');

TEST_FINISHED();
END_METHOD

METHOD PUBLIC Check_BYTE_TO_STRING_Max
VAR
	value : BYTE := DatatypeLimits.BYTE_MAX_VALUE;
	actual : STRING;
	converted : BOOL;
	equal : BOOL;
END_VAR
TEST('Check_BYTE_TO_STRING_Max');

// @TEST-RUN
converted := TryConvert_BYTE_TO_Destination(value, actual);
equal := actual = BYTE_TO_STRING(value);

// @TEST-ASSERT
AssertTrue(Condition := equal, Message := 'Did not convert BYTE to STRING correctly');
AssertTrue(Condition := converted, Message := 'Did not report BYTE to STRING conversion was successful');

TEST_FINISHED();
END_METHOD

METHOD PUBLIC Check_BYTE_TO_TIME_Min
VAR
	value : BYTE := DatatypeLimits.BYTE_MIN_VALUE;
	actual : TIME;
	converted : BOOL;
	equal : BOOL;
END_VAR
TEST('Check_BYTE_TO_TIME_Min');

// @TEST-RUN
converted := TryConvert_BYTE_TO_Destination(value, actual);
equal := actual = BYTE_TO_TIME(value);

// @TEST-ASSERT
AssertTrue(Condition := equal, Message := 'Did not convert BYTE to TIME correctly');
AssertTrue(Condition := converted, Message := 'Did not report BYTE to TIME conversion was successful');

TEST_FINISHED();
END_METHOD

METHOD PUBLIC Check_BYTE_TO_TIME_Max
VAR
	value : BYTE := DatatypeLimits.BYTE_MAX_VALUE;
	actual : TIME;
	converted : BOOL;
	equal : BOOL;
END_VAR
TEST('Check_BYTE_TO_TIME_Max');

// @TEST-RUN
converted := TryConvert_BYTE_TO_Destination(value, actual);
equal := actual = BYTE_TO_TIME(value);

// @TEST-ASSERT
AssertTrue(Condition := equal, Message := 'Did not convert BYTE to TIME correctly');
AssertTrue(Condition := converted, Message := 'Did not report BYTE to TIME conversion was successful');

TEST_FINISHED();
END_METHOD

METHOD PUBLIC Check_BYTE_TO_TOD_Min
VAR
	value : BYTE := DatatypeLimits.BYTE_MIN_VALUE;
	actual : TOD;
	converted : BOOL;
	equal : BOOL;
END_VAR
TEST('Check_BYTE_TO_TOD_Min');

// @TEST-RUN
converted := TryConvert_BYTE_TO_Destination(value, actual);
equal := actual = BYTE_TO_TOD(value);

// @TEST-ASSERT
AssertTrue(Condition := equal, Message := 'Did not convert BYTE to TOD correctly');
AssertTrue(Condition := converted, Message := 'Did not report BYTE to TOD conversion was successful');

TEST_FINISHED();
END_METHOD

METHOD PUBLIC Check_BYTE_TO_TOD_Max
VAR
	value : BYTE := DatatypeLimits.BYTE_MAX_VALUE;
	actual : TOD;
	converted : BOOL;
	equal : BOOL;
END_VAR
TEST('Check_BYTE_TO_TOD_Max');

// @TEST-RUN
converted := TryConvert_BYTE_TO_Destination(value, actual);
equal := actual = BYTE_TO_TOD(value);

// @TEST-ASSERT
AssertTrue(Condition := equal, Message := 'Did not convert BYTE to TOD correctly');
AssertTrue(Condition := converted, Message := 'Did not report BYTE to TOD conversion was successful');

TEST_FINISHED();
END_METHOD

METHOD PUBLIC Check_BYTE_TO_UDINT_Min
VAR
	value : BYTE := DatatypeLimits.BYTE_MIN_VALUE;
	actual : UDINT;
	converted : BOOL;
	equal : BOOL;
END_VAR
TEST('Check_BYTE_TO_UDINT_Min');

// @TEST-RUN
converted := TryConvert_BYTE_TO_Destination(value, actual);
equal := actual = BYTE_TO_UDINT(value);

// @TEST-ASSERT
AssertTrue(Condition := equal, Message := 'Did not convert BYTE to UDINT correctly');
AssertTrue(Condition := converted, Message := 'Did not report BYTE to UDINT conversion was successful');

TEST_FINISHED();
END_METHOD

METHOD PUBLIC Check_BYTE_TO_UDINT_Max
VAR
	value : BYTE := DatatypeLimits.BYTE_MAX_VALUE;
	actual : UDINT;
	converted : BOOL;
	equal : BOOL;
END_VAR
TEST('Check_BYTE_TO_UDINT_Max');

// @TEST-RUN
converted := TryConvert_BYTE_TO_Destination(value, actual);
equal := actual = BYTE_TO_UDINT(value);

// @TEST-ASSERT
AssertTrue(Condition := equal, Message := 'Did not convert BYTE to UDINT correctly');
AssertTrue(Condition := converted, Message := 'Did not report BYTE to UDINT conversion was successful');

TEST_FINISHED();
END_METHOD

METHOD PUBLIC Check_BYTE_TO_UINT_Min
VAR
	value : BYTE := DatatypeLimits.BYTE_MIN_VALUE;
	actual : UINT;
	converted : BOOL;
	equal : BOOL;
END_VAR
TEST('Check_BYTE_TO_UINT_Min');

// @TEST-RUN
converted := TryConvert_BYTE_TO_Destination(value, actual);
equal := actual = BYTE_TO_UINT(value);

// @TEST-ASSERT
AssertTrue(Condition := equal, Message := 'Did not convert BYTE to UINT correctly');
AssertTrue(Condition := converted, Message := 'Did not report BYTE to UINT conversion was successful');

TEST_FINISHED();
END_METHOD

METHOD PUBLIC Check_BYTE_TO_UINT_Max
VAR
	value : BYTE := DatatypeLimits.BYTE_MAX_VALUE;
	actual : UINT;
	converted : BOOL;
	equal : BOOL;
END_VAR
TEST('Check_BYTE_TO_UINT_Max');

// @TEST-RUN
converted := TryConvert_BYTE_TO_Destination(value, actual);
equal := actual = BYTE_TO_UINT(value);

// @TEST-ASSERT
AssertTrue(Condition := equal, Message := 'Did not convert BYTE to UINT correctly');
AssertTrue(Condition := converted, Message := 'Did not report BYTE to UINT conversion was successful');

TEST_FINISHED();
END_METHOD

METHOD PUBLIC Check_BYTE_TO_ULINT_Min
VAR
	value : BYTE := DatatypeLimits.BYTE_MIN_VALUE;
	actual : ULINT;
	converted : BOOL;
	equal : BOOL;
END_VAR
TEST('Check_BYTE_TO_ULINT_Min');

// @TEST-RUN
converted := TryConvert_BYTE_TO_Destination(value, actual);
equal := actual = BYTE_TO_ULINT(value);

// @TEST-ASSERT
AssertTrue(Condition := equal, Message := 'Did not convert BYTE to ULINT correctly');
AssertTrue(Condition := converted, Message := 'Did not report BYTE to ULINT conversion was successful');

TEST_FINISHED();
END_METHOD

METHOD PUBLIC Check_BYTE_TO_ULINT_Max
VAR
	value : BYTE := DatatypeLimits.BYTE_MAX_VALUE;
	actual : ULINT;
	converted : BOOL;
	equal : BOOL;
END_VAR
TEST('Check_BYTE_TO_ULINT_Max');

// @TEST-RUN
converted := TryConvert_BYTE_TO_Destination(value, actual);
equal := actual = BYTE_TO_ULINT(value);

// @TEST-ASSERT
AssertTrue(Condition := equal, Message := 'Did not convert BYTE to ULINT correctly');
AssertTrue(Condition := converted, Message := 'Did not report BYTE to ULINT conversion was successful');

TEST_FINISHED();
END_METHOD

METHOD PUBLIC Check_BYTE_TO_USINT_Min
VAR
	value : BYTE := DatatypeLimits.BYTE_MIN_VALUE;
	actual : USINT;
	converted : BOOL;
	equal : BOOL;
END_VAR
TEST('Check_BYTE_TO_USINT_Min');

// @TEST-RUN
converted := TryConvert_BYTE_TO_Destination(value, actual);
equal := actual = BYTE_TO_USINT(value);

// @TEST-ASSERT
AssertTrue(Condition := equal, Message := 'Did not convert BYTE to USINT correctly');
AssertTrue(Condition := converted, Message := 'Did not report BYTE to USINT conversion was successful');

TEST_FINISHED();
END_METHOD

METHOD PUBLIC Check_BYTE_TO_USINT_Max
VAR
	value : BYTE := DatatypeLimits.BYTE_MAX_VALUE;
	actual : USINT;
	converted : BOOL;
	equal : BOOL;
END_VAR
TEST('Check_BYTE_TO_USINT_Max');

// @TEST-RUN
converted := TryConvert_BYTE_TO_Destination(value, actual);
equal := actual = BYTE_TO_USINT(value);

// @TEST-ASSERT
AssertTrue(Condition := equal, Message := 'Did not convert BYTE to USINT correctly');
AssertTrue(Condition := converted, Message := 'Did not report BYTE to USINT conversion was successful');

TEST_FINISHED();
END_METHOD

METHOD PUBLIC Check_BYTE_TO_WORD_Min
VAR
	value : BYTE := DatatypeLimits.BYTE_MIN_VALUE;
	actual : WORD;
	converted : BOOL;
	equal : BOOL;
END_VAR
TEST('Check_BYTE_TO_WORD_Min');

// @TEST-RUN
converted := TryConvert_BYTE_TO_Destination(value, actual);
equal := actual = BYTE_TO_WORD(value);

// @TEST-ASSERT
AssertTrue(Condition := equal, Message := 'Did not convert BYTE to WORD correctly');
AssertTrue(Condition := converted, Message := 'Did not report BYTE to WORD conversion was successful');

TEST_FINISHED();
END_METHOD

METHOD PUBLIC Check_BYTE_TO_WORD_Max
VAR
	value : BYTE := DatatypeLimits.BYTE_MAX_VALUE;
	actual : WORD;
	converted : BOOL;
	equal : BOOL;
END_VAR
TEST('Check_BYTE_TO_WORD_Max');

// @TEST-RUN
converted := TryConvert_BYTE_TO_Destination(value, actual);
equal := actual = BYTE_TO_WORD(value);

// @TEST-ASSERT
AssertTrue(Condition := equal, Message := 'Did not convert BYTE to WORD correctly');
AssertTrue(Condition := converted, Message := 'Did not report BYTE to WORD conversion was successful');

TEST_FINISHED();
END_METHOD

END_FUNCTION_BLOCK

// ---- Tests/WORD_TO_TestSuite.TcPOU
FUNCTION_BLOCK PUBLIC WORD_TO_TestSuite EXTENDS TcUnit.FB_TestSuite
VAR
END_VAR

Check_WORD_TO_BOOL_Max();
Check_WORD_TO_BOOL_Min();
Check_WORD_TO_BYTE_Max();
Check_WORD_TO_BYTE_Min();
Check_WORD_TO_BYTE_TooHigh();
Check_WORD_TO_WORD_Max();
Check_WORD_TO_WORD_Min();
Check_WORD_TO_DWORD_Max();
Check_WORD_TO_DWORD_Min();
Check_WORD_TO_LWORD_Max();
Check_WORD_TO_LWORD_Min();
Check_WORD_TO_SINT_Max();
Check_WORD_TO_SINT_Min();
Check_WORD_TO_SINT_TooHigh();
Check_WORD_TO_INT_Max();
Check_WORD_TO_INT_Min();
Check_WORD_TO_INT_TooHigh();
Check_WORD_TO_DINT_Max();
Check_WORD_TO_DINT_Min();
Check_WORD_TO_LINT_Max();
Check_WORD_TO_LINT_Min();
Check_WORD_TO_USINT_Max();
Check_WORD_TO_USINT_Min();
Check_WORD_TO_USINT_TooHigh();
Check_WORD_TO_UINT_Max();
Check_WORD_TO_UINT_Min();
Check_WORD_TO_UDINT_Max();
Check_WORD_TO_UDINT_Min();
Check_WORD_TO_ULINT_Max();
Check_WORD_TO_ULINT_Min();
Check_WORD_TO_REAL_Max();
Check_WORD_TO_REAL_Min();
Check_WORD_TO_LREAL_Max();
Check_WORD_TO_LREAL_Min();
Check_WORD_TO_TIME_Max();
Check_WORD_TO_TIME_Min();
Check_WORD_TO_TOD_Max();
Check_WORD_TO_TOD_Min();
Check_WORD_TO_DATE_Max();
Check_WORD_TO_DATE_Min();
Check_WORD_TO_DT_Max();
Check_WORD_TO_DT_Min();
Check_WORD_TO_STRING_Max();
Check_WORD_TO_STRING_Min();

METHOD PUBLIC Check_WORD_TO_BOOL_Min
VAR
	value : WORD := DatatypeLimits.WORD_MIN_VALUE;
	actual : BOOL;
	converted : BOOL;
	equal : BOOL;
END_VAR
TEST('Check_WORD_TO_BOOL_Min');

// @TEST-RUN
converted := TryConvert_WORD_TO_Destination(value, actual);
equal := actual = WORD_TO_BOOL(value);

// @TEST-ASSERT
AssertTrue(Condition := equal, Message := 'Did not convert WORD to BOOL correctly');
AssertTrue(Condition := converted, Message := 'Did not report WORD to BOOL conversion was successful');

TEST_FINISHED();
END_METHOD

METHOD PUBLIC Check_WORD_TO_BOOL_Max
VAR
	value : WORD := DatatypeLimits.WORD_MAX_VALUE;
	actual : BOOL;
	converted : BOOL;
	equal : BOOL;
END_VAR
TEST('Check_WORD_TO_BOOL_Max');

// @TEST-RUN
converted := TryConvert_WORD_TO_Destination(value, actual);
equal := actual = WORD_TO_BOOL(value);

// @TEST-ASSERT
AssertTrue(Condition := equal, Message := 'Did not convert WORD to BOOL correctly');
AssertTrue(Condition := converted, Message := 'Did not report WORD to BOOL conversion was successful');

TEST_FINISHED();
END_METHOD

METHOD PUBLIC Check_WORD_TO_BYTE_Min
VAR
	value : WORD := DatatypeLimits.WORD_MIN_VALUE;
	actual : BYTE;
	converted : BOOL;
	equal : BOOL;
END_VAR
TEST('Check_WORD_TO_BYTE_Min');

// @TEST-RUN
converted := TryConvert_WORD_TO_Destination(value, actual);
equal := actual = WORD_TO_BYTE(value);

// @TEST-ASSERT
AssertTrue(Condition := equal, Message := 'Did not convert WORD to BYTE correctly');
AssertTrue(Condition := converted, Message := 'Did not report WORD to BYTE conversion was successful');

TEST_FINISHED();
END_METHOD

METHOD PUBLIC Check_WORD_TO_BYTE_TooHigh
VAR
	value : WORD := DatatypeLimits.WORD_MAX_VALUE;
	actual : BYTE;
	converted : BOOL;
END_VAR
TEST('Check_WORD_TO_BYTE_TooHigh');

// @TEST-RUN
converted := TryConvert_WORD_TO_Destination(value, actual);

// @TEST-ASSERT
AssertFalse(Condition := converted, Message := 'Did not report WORD to BYTE conversion was prevented');

TEST_FINISHED();
END_METHOD

METHOD PUBLIC Check_WORD_TO_BYTE_Max
VAR
	value : WORD := DatatypeLimits.MAX_VALUE_OF_WORD_WHICH_CAN_BE_HELD_IN_A_BYTE;
	actual : BYTE;
	converted : BOOL;
	equal : BOOL;
END_VAR
TEST('Check_WORD_TO_BYTE_Max');

// @TEST-RUN
converted := TryConvert_WORD_TO_Destination(value, actual);
equal := actual = WORD_TO_BYTE(value);

// @TEST-ASSERT
AssertTrue(Condition := equal, Message := 'Did not convert WORD to BYTE correctly');
AssertTrue(Condition := converted, Message := 'Did not report WORD to BYTE conversion was successful');

TEST_FINISHED();
END_METHOD

METHOD PUBLIC Check_WORD_TO_DATE_Min
VAR
	value : WORD := DatatypeLimits.WORD_MIN_VALUE;
	actual : DATE;
	converted : BOOL;
	equal : BOOL;
END_VAR
TEST('Check_WORD_TO_DATE_Min');

// @TEST-RUN
converted := TryConvert_WORD_TO_Destination(value, actual);
equal := actual = WORD_TO_DATE(value);

// @TEST-ASSERT
AssertTrue(Condition := equal, Message := 'Did not convert WORD to DATE correctly');
AssertTrue(Condition := converted, Message := 'Did not report WORD to DATE conversion was successful');

TEST_FINISHED();
END_METHOD

METHOD PUBLIC Check_WORD_TO_DATE_Max
VAR
	value : WORD := DatatypeLimits.WORD_MAX_VALUE;
	actual : DATE;
	converted : BOOL;
	equal : BOOL;
END_VAR
TEST('Check_WORD_TO_DATE_Max');

// @TEST-RUN
converted := TryConvert_WORD_TO_Destination(value, actual);
equal := actual = WORD_TO_DATE(value);

// @TEST-ASSERT
AssertTrue(Condition := equal, Message := 'Did not convert WORD to DATE correctly');
AssertTrue(Condition := converted, Message := 'Did not report WORD to DATE conversion was successful');

TEST_FINISHED();
END_METHOD

METHOD PUBLIC Check_WORD_TO_DINT_Min
VAR
	value : WORD := DatatypeLimits.WORD_MIN_VALUE;
	actual : DINT;
	converted : BOOL;
	equal : BOOL;
END_VAR
TEST('Check_WORD_TO_DINT_Min');

// @TEST-RUN
converted := TryConvert_WORD_TO_Destination(value, actual);
equal := actual = WORD_TO_DINT(value);

// @TEST-ASSERT
AssertTrue(Condition := equal, Message := 'Did not convert WORD to DINT correctly');
AssertTrue(Condition := converted, Message := 'Did not report WORD to DINT conversion was successful');

TEST_FINISHED();
END_METHOD

METHOD PUBLIC Check_WORD_TO_DINT_Max
VAR
	value : WORD := DatatypeLimits.WORD_MAX_VALUE;
	actual : DINT;
	converted : BOOL;
	equal : BOOL;
END_VAR
TEST('Check_WORD_TO_DINT_Max');

// @TEST-RUN
converted := TryConvert_WORD_TO_Destination(value, actual);
equal := actual = WORD_TO_DINT(value);

// @TEST-ASSERT
AssertTrue(Condition := equal, Message := 'Did not convert WORD to DINT correctly');
AssertTrue(Condition := converted, Message := 'Did not report WORD to DINT conversion was successful');

TEST_FINISHED();
END_METHOD

METHOD PUBLIC Check_WORD_TO_DT_Min
VAR
	value : WORD := DatatypeLimits.WORD_MIN_VALUE;
	actual : DT;
	converted : BOOL;
	equal : BOOL;
END_VAR
TEST('Check_WORD_TO_DT_Min');

// @TEST-RUN
converted := TryConvert_WORD_TO_Destination(value, actual);
equal := actual = WORD_TO_DT(value);

// @TEST-ASSERT
AssertTrue(Condition := equal, Message := 'Did not convert WORD to DT correctly');
AssertTrue(Condition := converted, Message := 'Did not report WORD to DT conversion was successful');

TEST_FINISHED();
END_METHOD

METHOD PUBLIC Check_WORD_TO_DT_Max
VAR
	value : WORD := DatatypeLimits.WORD_MAX_VALUE;
	actual : DT;
	converted : BOOL;
	equal : BOOL;
END_VAR
TEST('Check_WORD_TO_DT_Max');

// @TEST-RUN
converted := TryConvert_WORD_TO_Destination(value, actual);
equal := actual = WORD_TO_DT(value);

// @TEST-ASSERT
AssertTrue(Condition := equal, Message := 'Did not convert WORD to DT correctly');
AssertTrue(Condition := converted, Message := 'Did not report WORD to DT conversion was successful');

TEST_FINISHED();
END_METHOD

METHOD PUBLIC Check_WORD_TO_DWORD_Min
VAR
	value : WORD := DatatypeLimits.WORD_MIN_VALUE;
	actual : DWORD;
	converted : BOOL;
	equal : BOOL;
END_VAR
TEST('Check_WORD_TO_DWORD_Min');

// @TEST-RUN
converted := TryConvert_WORD_TO_Destination(value, actual);
equal := actual = WORD_TO_DWORD(value);

// @TEST-ASSERT
AssertTrue(Condition := equal, Message := 'Did not convert WORD to DWORD correctly');
AssertTrue(Condition := converted, Message := 'Did not report WORD to DWORD conversion was successful');

TEST_FINISHED();
END_METHOD

METHOD PUBLIC Check_WORD_TO_DWORD_Max
VAR
	value : WORD := DatatypeLimits.WORD_MAX_VALUE;
	actual : DWORD;
	converted : BOOL;
	equal : BOOL;
END_VAR
TEST('Check_WORD_TO_DWORD_Max');

// @TEST-RUN
converted := TryConvert_WORD_TO_Destination(value, actual);
equal := actual = WORD_TO_DWORD(value);

// @TEST-ASSERT
AssertTrue(Condition := equal, Message := 'Did not convert WORD to DWORD correctly');
AssertTrue(Condition := converted, Message := 'Did not report WORD to DWORD conversion was successful');

TEST_FINISHED();
END_METHOD

METHOD PUBLIC Check_WORD_TO_INT_Min
VAR
	value : WORD := DatatypeLimits.WORD_MIN_VALUE;
	actual : INT;
	converted : BOOL;
	equal : BOOL;
END_VAR
TEST('Check_WORD_TO_INT_Min');

// @TEST-RUN
converted := TryConvert_WORD_TO_Destination(value, actual);
equal := actual = WORD_TO_INT(value);

// @TEST-ASSERT
AssertTrue(Condition := equal, Message := 'Did not convert WORD to INT correctly');
AssertTrue(Condition := converted, Message := 'Did not report WORD to INT conversion was successful');

TEST_FINISHED();
END_METHOD

METHOD PUBLIC Check_WORD_TO_INT_TooHigh
VAR
	value : WORD := DatatypeLimits.WORD_MAX_VALUE;
	actual : INT;
	converted : BOOL;
END_VAR
TEST('Check_WORD_TO_INT_TooHigh');

// @TEST-RUN
converted := TryConvert_WORD_TO_Destination(value, actual);

// @TEST-ASSERT
AssertFalse(Condition := converted, Message := 'Did not report WORD to INT conversion was prevented');

TEST_FINISHED();
END_METHOD

METHOD PUBLIC Check_WORD_TO_INT_Max
VAR
	value : WORD := DatatypeLimits.MAX_VALUE_OF_WORD_WHICH_CAN_BE_HELD_IN_A_INT;
	actual : INT;
	converted : BOOL;
	equal : BOOL;
END_VAR
TEST('Check_WORD_TO_INT_Max');

// @TEST-RUN
converted := TryConvert_WORD_TO_Destination(value, actual);
equal := actual = WORD_TO_INT(value);

// @TEST-ASSERT
AssertTrue(Condition := equal, Message := 'Did not convert WORD to INT correctly');
AssertTrue(Condition := converted, Message := 'Did not report WORD to INT conversion was successful');

TEST_FINISHED();
END_METHOD

METHOD PUBLIC Check_WORD_TO_LINT_Min
VAR
	value : WORD := DatatypeLimits.WORD_MIN_VALUE;
	actual : LINT;
	converted : BOOL;
	equal : BOOL;
END_VAR
TEST('Check_WORD_TO_LINT_Min');

// @TEST-RUN
converted := TryConvert_WORD_TO_Destination(value, actual);
equal := actual = WORD_TO_LINT(value);

// @TEST-ASSERT
AssertTrue(Condition := equal, Message := 'Did not convert WORD to LINT correctly');
AssertTrue(Condition := converted, Message := 'Did not report WORD to LINT conversion was successful');

TEST_FINISHED();
END_METHOD

METHOD PUBLIC Check_WORD_TO_LINT_Max
VAR
	value : WORD := DatatypeLimits.WORD_MAX_VALUE;
	actual : LINT;
	converted : BOOL;
	equal : BOOL;
END_VAR
TEST('Check_WORD_TO_LINT_Max');

// @TEST-RUN
converted := TryConvert_WORD_TO_Destination(value, actual);
equal := actual = WORD_TO_LINT(value);

// @TEST-ASSERT
AssertTrue(Condition := equal, Message := 'Did not convert WORD to LINT correctly');
AssertTrue(Condition := converted, Message := 'Did not report WORD to LINT conversion was successful');

TEST_FINISHED();
END_METHOD

METHOD PUBLIC Check_WORD_TO_LREAL_Min
VAR
	value : WORD := DatatypeLimits.WORD_MIN_VALUE;
	actual : LREAL;
	converted : BOOL;
	equal : BOOL;
END_VAR
TEST('Check_WORD_TO_LREAL_Min');

// @TEST-RUN
converted := TryConvert_WORD_TO_Destination(value, actual);
equal := actual = WORD_TO_LREAL(value);

// @TEST-ASSERT
AssertTrue(Condition := equal, Message := 'Did not convert WORD to LREAL correctly');
AssertTrue(Condition := converted, Message := 'Did not report WORD to LREAL conversion was successful');

TEST_FINISHED();
END_METHOD

METHOD PUBLIC Check_WORD_TO_LREAL_Max
VAR
	value : WORD := DatatypeLimits.WORD_MAX_VALUE;
	actual : LREAL;
	converted : BOOL;
	equal : BOOL;
END_VAR
TEST('Check_WORD_TO_LREAL_Max');

// @TEST-RUN
converted := TryConvert_WORD_TO_Destination(value, actual);
equal := actual = WORD_TO_LREAL(value);

// @TEST-ASSERT
AssertTrue(Condition := equal, Message := 'Did not convert WORD to LREAL correctly');
AssertTrue(Condition := converted, Message := 'Did not report WORD to LREAL conversion was successful');

TEST_FINISHED();
END_METHOD

METHOD PUBLIC Check_WORD_TO_LWORD_Min
VAR
	value : WORD := DatatypeLimits.WORD_MIN_VALUE;
	actual : LWORD;
	converted : BOOL;
	equal : BOOL;
END_VAR
TEST('Check_WORD_TO_LWORD_Min');

// @TEST-RUN
converted := TryConvert_WORD_TO_Destination(value, actual);
equal := actual = WORD_TO_LWORD(value);

// @TEST-ASSERT
AssertTrue(Condition := equal, Message := 'Did not convert WORD to LWORD correctly');
AssertTrue(Condition := converted, Message := 'Did not report WORD to LWORD conversion was successful');

TEST_FINISHED();
END_METHOD

METHOD PUBLIC Check_WORD_TO_LWORD_Max
VAR
	value : WORD := DatatypeLimits.WORD_MAX_VALUE;
	actual : LWORD;
	converted : BOOL;
	equal : BOOL;
END_VAR
TEST('Check_WORD_TO_LWORD_Max');

// @TEST-RUN
converted := TryConvert_WORD_TO_Destination(value, actual);
equal := actual = WORD_TO_LWORD(value);

// @TEST-ASSERT
AssertTrue(Condition := equal, Message := 'Did not convert WORD to LWORD correctly');
AssertTrue(Condition := converted, Message := 'Did not report WORD to LWORD conversion was successful');

TEST_FINISHED();
END_METHOD

METHOD PUBLIC Check_WORD_TO_REAL_Min
VAR
	value : WORD := DatatypeLimits.WORD_MIN_VALUE;
	actual : REAL;
	converted : BOOL;
	equal : BOOL;
END_VAR
TEST('Check_WORD_TO_REAL_Min');

// @TEST-RUN
converted := TryConvert_WORD_TO_Destination(value, actual);
equal := actual = WORD_TO_REAL(value);

// @TEST-ASSERT
AssertTrue(Condition := equal, Message := 'Did not convert WORD to REAL correctly');
AssertTrue(Condition := converted, Message := 'Did not report WORD to REAL conversion was successful');

TEST_FINISHED();
END_METHOD

METHOD PUBLIC Check_WORD_TO_REAL_Max
VAR
	value : WORD := DatatypeLimits.WORD_MAX_VALUE;
	actual : REAL;
	converted : BOOL;
	equal : BOOL;
END_VAR
TEST('Check_WORD_TO_REAL_Max');

// @TEST-RUN
converted := TryConvert_WORD_TO_Destination(value, actual);
equal := actual = WORD_TO_REAL(value);

// @TEST-ASSERT
AssertTrue(Condition := equal, Message := 'Did not convert WORD to REAL correctly');
AssertTrue(Condition := converted, Message := 'Did not report WORD to REAL conversion was successful');

TEST_FINISHED();
END_METHOD

METHOD PUBLIC Check_WORD_TO_SINT_Min
VAR
	value : WORD := DatatypeLimits.WORD_MIN_VALUE;
	actual : SINT;
	converted : BOOL;
	equal : BOOL;
END_VAR
TEST('Check_WORD_TO_SINT_Min');

// @TEST-RUN
converted := TryConvert_WORD_TO_Destination(value, actual);
equal := actual = WORD_TO_SINT(value);

// @TEST-ASSERT
AssertTrue(Condition := equal, Message := 'Did not convert WORD to SINT correctly');
AssertTrue(Condition := converted, Message := 'Did not report WORD to SINT conversion was successful');

TEST_FINISHED();
END_METHOD

METHOD PUBLIC Check_WORD_TO_SINT_TooHigh
VAR
	value : WORD := DatatypeLimits.WORD_MAX_VALUE;
	actual : SINT;
	converted : BOOL;
END_VAR
TEST('Check_WORD_TO_SINT_TooHigh');

// @TEST-RUN
converted := TryConvert_WORD_TO_Destination(value, actual);

// @TEST-ASSERT
AssertFalse(Condition := converted, Message := 'Did not report WORD to SINT conversion was prevented');

TEST_FINISHED();
END_METHOD

METHOD PUBLIC Check_WORD_TO_SINT_Max
VAR
	value : WORD := DatatypeLimits.MAX_VALUE_OF_WORD_WHICH_CAN_BE_HELD_IN_A_SINT;
	actual : SINT;
	converted : BOOL;
	equal : BOOL;
END_VAR
TEST('Check_WORD_TO_SINT_Max');

// @TEST-RUN
converted := TryConvert_WORD_TO_Destination(value, actual);
equal := actual = WORD_TO_SINT(value);

// @TEST-ASSERT
AssertTrue(Condition := equal, Message := 'Did not convert WORD to SINT correctly');
AssertTrue(Condition := converted, Message := 'Did not report WORD to SINT conversion was successful');

TEST_FINISHED();
END_METHOD

METHOD PUBLIC Check_WORD_TO_STRING_Min
VAR
	value : WORD := DatatypeLimits.WORD_MIN_VALUE;
	actual : STRING;
	converted : BOOL;
	equal : BOOL;
END_VAR
TEST('Check_WORD_TO_STRING_Min');

// @TEST-RUN
converted := TryConvert_WORD_TO_Destination(value, actual);
equal := actual = WORD_TO_STRING(value);

// @TEST-ASSERT
AssertTrue(Condition := equal, Message := 'Did not convert WORD to STRING correctly');
AssertTrue(Condition := converted, Message := 'Did not report WORD to STRING conversion was successful');

TEST_FINISHED();
END_METHOD

METHOD PUBLIC Check_WORD_TO_STRING_Max
VAR
	value : WORD := DatatypeLimits.WORD_MAX_VALUE;
	actual : STRING;
	converted : BOOL;
	equal : BOOL;
END_VAR
TEST('Check_WORD_TO_STRING_Max');

// @TEST-RUN
converted := TryConvert_WORD_TO_Destination(value, actual);
equal := actual = WORD_TO_STRING(value);

// @TEST-ASSERT
AssertTrue(Condition := equal, Message := 'Did not convert WORD to STRING correctly');
AssertTrue(Condition := converted, Message := 'Did not report WORD to STRING conversion was successful');

TEST_FINISHED();
END_METHOD

METHOD PUBLIC Check_WORD_TO_TIME_Min
VAR
	value : WORD := DatatypeLimits.WORD_MIN_VALUE;
	actual : TIME;
	converted : BOOL;
	equal : BOOL;
END_VAR
TEST('Check_WORD_TO_TIME_Min');

// @TEST-RUN
converted := TryConvert_WORD_TO_Destination(value, actual);
equal := actual = WORD_TO_TIME(value);

// @TEST-ASSERT
AssertTrue(Condition := equal, Message := 'Did not convert WORD to TIME correctly');
AssertTrue(Condition := converted, Message := 'Did not report WORD to TIME conversion was successful');

TEST_FINISHED();
END_METHOD

METHOD PUBLIC Check_WORD_TO_TIME_Max
VAR
	value : WORD := DatatypeLimits.WORD_MAX_VALUE;
	actual : TIME;
	converted : BOOL;
	equal : BOOL;
END_VAR
TEST('Check_WORD_TO_TIME_Max');

// @TEST-RUN
converted := TryConvert_WORD_TO_Destination(value, actual);
equal := actual = WORD_TO_TIME(value);

// @TEST-ASSERT
AssertTrue(Condition := equal, Message := 'Did not convert WORD to TIME correctly');
AssertTrue(Condition := converted, Message := 'Did not report WORD to TIME conversion was successful');

TEST_FINISHED();
END_METHOD

METHOD PUBLIC Check_WORD_TO_TOD_Min
VAR
	value : WORD := DatatypeLimits.WORD_MIN_VALUE;
	actual : TOD;
	converted : BOOL;
	equal : BOOL;
END_VAR
TEST('Check_WORD_TO_TOD_Min');

// @TEST-RUN
converted := TryConvert_WORD_TO_Destination(value, actual);
equal := actual = WORD_TO_TOD(value);

// @TEST-ASSERT
AssertTrue(Condition := equal, Message := 'Did not convert WORD to TOD correctly');
AssertTrue(Condition := converted, Message := 'Did not report WORD to TOD conversion was successful');

TEST_FINISHED();
END_METHOD

METHOD PUBLIC Check_WORD_TO_TOD_Max
VAR
	value : WORD := DatatypeLimits.WORD_MAX_VALUE;
	actual : TOD;
	converted : BOOL;
	equal : BOOL;
END_VAR
TEST('Check_WORD_TO_TOD_Max');

// @TEST-RUN
converted := TryConvert_WORD_TO_Destination(value, actual);
equal := actual = WORD_TO_TOD(value);

// @TEST-ASSERT
AssertTrue(Condition := equal, Message := 'Did not convert WORD to TOD correctly');
AssertTrue(Condition := converted, Message := 'Did not report WORD to TOD conversion was successful');

TEST_FINISHED();
END_METHOD

METHOD PUBLIC Check_WORD_TO_UDINT_Min
VAR
	value : WORD := DatatypeLimits.WORD_MIN_VALUE;
	actual : UDINT;
	converted : BOOL;
	equal : BOOL;
END_VAR
TEST('Check_WORD_TO_UDINT_Min');

// @TEST-RUN
converted := TryConvert_WORD_TO_Destination(value, actual);
equal := actual = WORD_TO_UDINT(value);

// @TEST-ASSERT
AssertTrue(Condition := equal, Message := 'Did not convert WORD to UDINT correctly');
AssertTrue(Condition := converted, Message := 'Did not report WORD to UDINT conversion was successful');

TEST_FINISHED();
END_METHOD

METHOD PUBLIC Check_WORD_TO_UDINT_Max
VAR
	value : WORD := DatatypeLimits.WORD_MAX_VALUE;
	actual : UDINT;
	converted : BOOL;
	equal : BOOL;
END_VAR
TEST('Check_WORD_TO_UDINT_Max');

// @TEST-RUN
converted := TryConvert_WORD_TO_Destination(value, actual);
equal := actual = WORD_TO_UDINT(value);

// @TEST-ASSERT
AssertTrue(Condition := equal, Message := 'Did not convert WORD to UDINT correctly');
AssertTrue(Condition := converted, Message := 'Did not report WORD to UDINT conversion was successful');

TEST_FINISHED();
END_METHOD

METHOD PUBLIC Check_WORD_TO_UINT_Min
VAR
	value : WORD := DatatypeLimits.WORD_MIN_VALUE;
	actual : UINT;
	converted : BOOL;
	equal : BOOL;
END_VAR
TEST('Check_WORD_TO_UINT_Min');

// @TEST-RUN
converted := TryConvert_WORD_TO_Destination(value, actual);
equal := actual = WORD_TO_UINT(value);

// @TEST-ASSERT
AssertTrue(Condition := equal, Message := 'Did not convert WORD to UINT correctly');
AssertTrue(Condition := converted, Message := 'Did not report WORD to UINT conversion was successful');

TEST_FINISHED();
END_METHOD

METHOD PUBLIC Check_WORD_TO_UINT_Max
VAR
	value : WORD := DatatypeLimits.WORD_MAX_VALUE;
	actual : UINT;
	converted : BOOL;
	equal : BOOL;
END_VAR
TEST('Check_WORD_TO_UINT_Max');

// @TEST-RUN
converted := TryConvert_WORD_TO_Destination(value, actual);
equal := actual = WORD_TO_UINT(value);

// @TEST-ASSERT
AssertTrue(Condition := equal, Message := 'Did not convert WORD to UINT correctly');
AssertTrue(Condition := converted, Message := 'Did not report WORD to UINT conversion was successful');

TEST_FINISHED();
END_METHOD

METHOD PUBLIC Check_WORD_TO_ULINT_Min
VAR
	value : WORD := DatatypeLimits.WORD_MIN_VALUE;
	actual : ULINT;
	converted : BOOL;
	equal : BOOL;
END_VAR
TEST('Check_WORD_TO_ULINT_Min');

// @TEST-RUN
converted := TryConvert_WORD_TO_Destination(value, actual);
equal := actual = WORD_TO_ULINT(value);

// @TEST-ASSERT
AssertTrue(Condition := equal, Message := 'Did not convert WORD to ULINT correctly');
AssertTrue(Condition := converted, Message := 'Did not report WORD to ULINT conversion was successful');

TEST_FINISHED();
END_METHOD

METHOD PUBLIC Check_WORD_TO_ULINT_Max
VAR
	value : WORD := DatatypeLimits.WORD_MAX_VALUE;
	actual : ULINT;
	converted : BOOL;
	equal : BOOL;
END_VAR
TEST('Check_WORD_TO_ULINT_Max');

// @TEST-RUN
converted := TryConvert_WORD_TO_Destination(value, actual);
equal := actual = WORD_TO_ULINT(value);

// @TEST-ASSERT
AssertTrue(Condition := equal, Message := 'Did not convert WORD to ULINT correctly');
AssertTrue(Condition := converted, Message := 'Did not report WORD to ULINT conversion was successful');

TEST_FINISHED();
END_METHOD

METHOD PUBLIC Check_WORD_TO_USINT_Min
VAR
	value : WORD := DatatypeLimits.WORD_MIN_VALUE;
	actual : USINT;
	converted : BOOL;
	equal : BOOL;
END_VAR
TEST('Check_WORD_TO_USINT_Min');

// @TEST-RUN
converted := TryConvert_WORD_TO_Destination(value, actual);
equal := actual = WORD_TO_USINT(value);

// @TEST-ASSERT
AssertTrue(Condition := equal, Message := 'Did not convert WORD to USINT correctly');
AssertTrue(Condition := converted, Message := 'Did not report WORD to USINT conversion was successful');

TEST_FINISHED();
END_METHOD

METHOD PUBLIC Check_WORD_TO_USINT_TooHigh
VAR
	value : WORD := DatatypeLimits.WORD_MAX_VALUE;
	actual : USINT;
	converted : BOOL;
END_VAR
TEST('Check_WORD_TO_USINT_TooHigh');

// @TEST-RUN
converted := TryConvert_WORD_TO_Destination(value, actual);

// @TEST-ASSERT
AssertFalse(Condition := converted, Message := 'Did not report WORD to USINT conversion was prevented');

TEST_FINISHED();
END_METHOD

METHOD PUBLIC Check_WORD_TO_USINT_Max
VAR
	value : WORD := DatatypeLimits.MAX_VALUE_OF_WORD_WHICH_CAN_BE_HELD_IN_A_USINT;
	actual : USINT;
	converted : BOOL;
	equal : BOOL;
END_VAR
TEST('Check_WORD_TO_USINT_Max');

// @TEST-RUN
converted := TryConvert_WORD_TO_Destination(value, actual);
equal := actual = WORD_TO_USINT(value);

// @TEST-ASSERT
AssertTrue(Condition := equal, Message := 'Did not convert WORD to USINT correctly');
AssertTrue(Condition := converted, Message := 'Did not report WORD to USINT conversion was successful');

TEST_FINISHED();
END_METHOD

METHOD PUBLIC Check_WORD_TO_WORD_Min
VAR
	value : WORD := DatatypeLimits.WORD_MIN_VALUE;
	actual : WORD;
	converted : BOOL;
	equal : BOOL;
END_VAR
TEST('Check_WORD_TO_WORD_Min');

// @TEST-RUN
converted := TryConvert_WORD_TO_Destination(value, actual);
equal := actual = value;

// @TEST-ASSERT
AssertTrue(Condition := equal, Message := 'Did not convert WORD to WORD correctly');
AssertTrue(Condition := converted, Message := 'Did not report WORD to WORD conversion was successful');

TEST_FINISHED();
END_METHOD

METHOD PUBLIC Check_WORD_TO_WORD_Max
VAR
	value : WORD := DatatypeLimits.WORD_MAX_VALUE;
	actual : WORD;
	converted : BOOL;
	equal : BOOL;
END_VAR
TEST('Check_WORD_TO_WORD_Max');

// @TEST-RUN
converted := TryConvert_WORD_TO_Destination(value, actual);
equal := actual = value;

// @TEST-ASSERT
AssertTrue(Condition := equal, Message := 'Did not convert WORD to WORD correctly');
AssertTrue(Condition := converted, Message := 'Did not report WORD to WORD conversion was successful');

TEST_FINISHED();
END_METHOD

END_FUNCTION_BLOCK

// ---- Tests/DWORD_TO_TestSuite.TcPOU
FUNCTION_BLOCK PUBLIC DWORD_TO_TestSuite EXTENDS TcUnit.FB_TestSuite
VAR
END_VAR

Check_DWORD_TO_BOOL_Max();
Check_DWORD_TO_BOOL_Min();
Check_DWORD_TO_BYTE_Max();
Check_DWORD_TO_BYTE_Min();
Check_DWORD_TO_BYTE_TooHigh();
Check_DWORD_TO_WORD_Max();
Check_DWORD_TO_WORD_Min();
Check_DWORD_TO_WORD_TooHigh();
Check_DWORD_TO_DWORD_Max();
Check_DWORD_TO_DWORD_Min();
Check_DWORD_TO_LWORD_Max();
Check_DWORD_TO_LWORD_Min();
Check_DWORD_TO_SINT_Max();
Check_DWORD_TO_SINT_Min();
Check_DWORD_TO_SINT_TooHigh();
Check_DWORD_TO_INT_Max();
Check_DWORD_TO_INT_Min();
Check_DWORD_TO_INT_TooHigh();
Check_DWORD_TO_DINT_Max();
Check_DWORD_TO_DINT_Min();
Check_DWORD_TO_DINT_TooHigh();
Check_DWORD_TO_LINT_Max();
Check_DWORD_TO_LINT_Min();
Check_DWORD_TO_USINT_Max();
Check_DWORD_TO_USINT_Min();
Check_DWORD_TO_USINT_TooHigh();
Check_DWORD_TO_UINT_Max();
Check_DWORD_TO_UINT_Min();
Check_DWORD_TO_UINT_TooHigh();
Check_DWORD_TO_UDINT_Max();
Check_DWORD_TO_UDINT_Min();
Check_DWORD_TO_ULINT_Max();
Check_DWORD_TO_ULINT_Min();
Check_DWORD_TO_REAL_Max();
Check_DWORD_TO_REAL_Min();
Check_DWORD_TO_LREAL_Max();
Check_DWORD_TO_LREAL_Min();
Check_DWORD_TO_TIME_Max();
Check_DWORD_TO_TIME_Min();
Check_DWORD_TO_TOD_Max();
Check_DWORD_TO_TOD_Min();
Check_DWORD_TO_TOD_TooHigh();
Check_DWORD_TO_DATE_Max();
Check_DWORD_TO_DATE_Min();
Check_DWORD_TO_DT_Max();
Check_DWORD_TO_DT_Min();
Check_DWORD_TO_STRING_Max();
Check_DWORD_TO_STRING_Min();

METHOD PUBLIC Check_DWORD_TO_BOOL_Min
VAR
	value : DWORD := DatatypeLimits.DWORD_MIN_VALUE;
	actual : BOOL;
	converted : BOOL;
	equal : BOOL;
END_VAR
TEST('Check_DWORD_TO_BOOL_Min');

// @TEST-RUN
converted := TryConvert_DWORD_TO_Destination(value, actual);
equal := actual = DWORD_TO_BOOL(value);

// @TEST-ASSERT
AssertTrue(Condition := equal, Message := 'Did not convert DWORD to BOOL correctly');
AssertTrue(Condition := converted, Message := 'Did not report DWORD to BOOL conversion was successful');

TEST_FINISHED();
END_METHOD

METHOD PUBLIC Check_DWORD_TO_BOOL_Max
VAR
	value : DWORD := DatatypeLimits.DWORD_MAX_VALUE;
	actual : BOOL;
	converted : BOOL;
	equal : BOOL;
END_VAR
TEST('Check_DWORD_TO_BOOL_Max');

// @TEST-RUN
converted := TryConvert_DWORD_TO_Destination(value, actual);
equal := actual = DWORD_TO_BOOL(value);

// @TEST-ASSERT
AssertTrue(Condition := equal, Message := 'Did not convert DWORD to BOOL correctly');
AssertTrue(Condition := converted, Message := 'Did not report DWORD to BOOL conversion was successful');

TEST_FINISHED();
END_METHOD

METHOD PUBLIC Check_DWORD_TO_BYTE_Min
VAR
	value : DWORD := DatatypeLimits.DWORD_MIN_VALUE;
	actual : BYTE;
	converted : BOOL;
	equal : BOOL;
END_VAR
TEST('Check_DWORD_TO_BYTE_Min');

// @TEST-RUN
converted := TryConvert_DWORD_TO_Destination(value, actual);
equal := actual = DWORD_TO_BYTE(value);

// @TEST-ASSERT
AssertTrue(Condition := equal, Message := 'Did not convert DWORD to BYTE correctly');
AssertTrue(Condition := converted, Message := 'Did not report DWORD to BYTE conversion was successful');

TEST_FINISHED();
END_METHOD

METHOD PUBLIC Check_DWORD_TO_BYTE_TooHigh
VAR
	value : DWORD := DatatypeLimits.DWORD_MAX_VALUE;
	actual : BYTE;
	converted : BOOL;
END_VAR
TEST('Check_DWORD_TO_BYTE_TooHigh');

// @TEST-RUN
converted := TryConvert_DWORD_TO_Destination(value, actual);

// @TEST-ASSERT
AssertFalse(Condition := converted, Message := 'Did not report DWORD to BYTE conversion was prevented');

TEST_FINISHED();
END_METHOD

METHOD PUBLIC Check_DWORD_TO_BYTE_Max
VAR
	value : DWORD := DatatypeLimits.MAX_VALUE_OF_DWORD_WHICH_CAN_BE_HELD_IN_A_BYTE;
	actual : BYTE;
	converted : BOOL;
	equal : BOOL;
END_VAR
TEST('Check_DWORD_TO_BYTE_Max');

// @TEST-RUN
converted := TryConvert_DWORD_TO_Destination(value, actual);
equal := actual = DWORD_TO_BYTE(value);

// @TEST-ASSERT
AssertTrue(Condition := equal, Message := 'Did not convert DWORD to BYTE correctly');
AssertTrue(Condition := converted, Message := 'Did not report DWORD to BYTE conversion was successful');

TEST_FINISHED();
END_METHOD

METHOD PUBLIC Check_DWORD_TO_DATE_Min
VAR
	value : DWORD := DatatypeLimits.DWORD_MIN_VALUE;
	actual : DATE;
	converted : BOOL;
	equal : BOOL;
END_VAR
TEST('Check_DWORD_TO_DATE_Min');

// @TEST-RUN
converted := TryConvert_DWORD_TO_Destination(value, actual);
equal := actual = DWORD_TO_DATE(value);

// @TEST-ASSERT
AssertTrue(Condition := equal, Message := 'Did not convert DWORD to DATE correctly');
AssertTrue(Condition := converted, Message := 'Did not report DWORD to DATE conversion was successful');

TEST_FINISHED();
END_METHOD

METHOD PUBLIC Check_DWORD_TO_DATE_Max
VAR
	value : DWORD := DatatypeLimits.DWORD_MAX_VALUE;
	actual : DATE;
	converted : BOOL;
	equal : BOOL;
END_VAR
TEST('Check_DWORD_TO_DATE_Max');

// @TEST-RUN
converted := TryConvert_DWORD_TO_Destination(value, actual);
equal := actual = DWORD_TO_DATE(value);

// @TEST-ASSERT
AssertTrue(Condition := equal, Message := 'Did not convert DWORD to DATE correctly');
AssertTrue(Condition := converted, Message := 'Did not report DWORD to DATE conversion was successful');

TEST_FINISHED();
END_METHOD

METHOD PUBLIC Check_DWORD_TO_DINT_Min
VAR
	value : DWORD := DatatypeLimits.DWORD_MIN_VALUE;
	actual : DINT;
	converted : BOOL;
	equal : BOOL;
END_VAR
TEST('Check_DWORD_TO_DINT_Min');

// @TEST-RUN
converted := TryConvert_DWORD_TO_Destination(value, actual);
equal := actual = DWORD_TO_DINT(value);

// @TEST-ASSERT
AssertTrue(Condition := equal, Message := 'Did not convert DWORD to DINT correctly');
AssertTrue(Condition := converted, Message := 'Did not report DWORD to DINT conversion was successful');

TEST_FINISHED();
END_METHOD

METHOD PUBLIC Check_DWORD_TO_DINT_TooHigh
VAR
	value : DWORD := DatatypeLimits.DWORD_MAX_VALUE;
	actual : DINT;
	converted : BOOL;
END_VAR
TEST('Check_DWORD_TO_DINT_TooHigh');

// @TEST-RUN
converted := TryConvert_DWORD_TO_Destination(value, actual);

// @TEST-ASSERT
AssertFalse(Condition := converted, Message := 'Did not report DWORD to DINT conversion was prevented');

TEST_FINISHED();
END_METHOD

METHOD PUBLIC Check_DWORD_TO_DINT_Max
VAR
	value : DWORD := DatatypeLimits.MAX_VALUE_OF_DWORD_WHICH_CAN_BE_HELD_IN_A_DINT;
	actual : DINT;
	converted : BOOL;
	equal : BOOL;
END_VAR
TEST('Check_DWORD_TO_DINT_Max');

// @TEST-RUN
converted := TryConvert_DWORD_TO_Destination(value, actual);
equal := actual = DWORD_TO_DINT(value);

// @TEST-ASSERT
AssertTrue(Condition := equal, Message := 'Did not convert DWORD to DINT correctly');
AssertTrue(Condition := converted, Message := 'Did not report DWORD to DINT conversion was successful');

TEST_FINISHED();
END_METHOD

METHOD PUBLIC Check_DWORD_TO_DT_Min
VAR
	value : DWORD := DatatypeLimits.DWORD_MIN_VALUE;
	actual : DT;
	converted : BOOL;
	equal : BOOL;
END_VAR
TEST('Check_DWORD_TO_DT_Min');

// @TEST-RUN
converted := TryConvert_DWORD_TO_Destination(value, actual);
equal := actual = DWORD_TO_DT(value);

// @TEST-ASSERT
AssertTrue(Condition := equal, Message := 'Did not convert DWORD to DT correctly');
AssertTrue(Condition := converted, Message := 'Did not report DWORD to DT conversion was successful');

TEST_FINISHED();
END_METHOD

METHOD PUBLIC Check_DWORD_TO_DT_Max
VAR
	value : DWORD := DatatypeLimits.DWORD_MAX_VALUE;
	actual : DT;
	converted : BOOL;
	equal : BOOL;
END_VAR
TEST('Check_DWORD_TO_DT_Max');

// @TEST-RUN
converted := TryConvert_DWORD_TO_Destination(value, actual);
equal := actual = DWORD_TO_DT(value);

// @TEST-ASSERT
AssertTrue(Condition := equal, Message := 'Did not convert DWORD to DT correctly');
AssertTrue(Condition := converted, Message := 'Did not report DWORD to DT conversion was successful');

TEST_FINISHED();
END_METHOD

METHOD PUBLIC Check_DWORD_TO_DWORD_Min
VAR
	value : DWORD := DatatypeLimits.DWORD_MIN_VALUE;
	actual : DWORD;
	converted : BOOL;
	equal : BOOL;
END_VAR
TEST('Check_DWORD_TO_DWORD_Min');

// @TEST-RUN
converted := TryConvert_DWORD_TO_Destination(value, actual);
equal := actual = value;

// @TEST-ASSERT
AssertTrue(Condition := equal, Message := 'Did not convert DWORD to DWORD correctly');
AssertTrue(Condition := converted, Message := 'Did not report DWORD to DWORD conversion was successful');

TEST_FINISHED();
END_METHOD

METHOD PUBLIC Check_DWORD_TO_DWORD_Max
VAR
	value : DWORD := DatatypeLimits.DWORD_MAX_VALUE;
	actual : DWORD;
	converted : BOOL;
	equal : BOOL;
END_VAR
TEST('Check_DWORD_TO_DWORD_Max');

// @TEST-RUN
converted := TryConvert_DWORD_TO_Destination(value, actual);
equal := actual = value;

// @TEST-ASSERT
AssertTrue(Condition := equal, Message := 'Did not convert DWORD to DWORD correctly');
AssertTrue(Condition := converted, Message := 'Did not report DWORD to DWORD conversion was successful');

TEST_FINISHED();
END_METHOD

METHOD PUBLIC Check_DWORD_TO_INT_Min
VAR
	value : DWORD := DatatypeLimits.DWORD_MIN_VALUE;
	actual : INT;
	converted : BOOL;
	equal : BOOL;
END_VAR
TEST('Check_DWORD_TO_INT_Min');

// @TEST-RUN
converted := TryConvert_DWORD_TO_Destination(value, actual);
equal := actual = DWORD_TO_INT(value);

// @TEST-ASSERT
AssertTrue(Condition := equal, Message := 'Did not convert DWORD to INT correctly');
AssertTrue(Condition := converted, Message := 'Did not report DWORD to INT conversion was successful');

TEST_FINISHED();
END_METHOD

METHOD PUBLIC Check_DWORD_TO_INT_TooHigh
VAR
	value : DWORD := DatatypeLimits.DWORD_MAX_VALUE;
	actual : INT;
	converted : BOOL;
END_VAR
TEST('Check_DWORD_TO_INT_TooHigh');

// @TEST-RUN
converted := TryConvert_DWORD_TO_Destination(value, actual);

// @TEST-ASSERT
AssertFalse(Condition := converted, Message := 'Did not report DWORD to INT conversion was prevented');

TEST_FINISHED();
END_METHOD

METHOD PUBLIC Check_DWORD_TO_INT_Max
VAR
	value : DWORD := DatatypeLimits.MAX_VALUE_OF_DWORD_WHICH_CAN_BE_HELD_IN_A_INT;
	actual : INT;
	converted : BOOL;
	equal : BOOL;
END_VAR
TEST('Check_DWORD_TO_INT_Max');

// @TEST-RUN
converted := TryConvert_DWORD_TO_Destination(value, actual);
equal := actual = DWORD_TO_INT(value);

// @TEST-ASSERT
AssertTrue(Condition := equal, Message := 'Did not convert DWORD to INT correctly');
AssertTrue(Condition := converted, Message := 'Did not report DWORD to INT conversion was successful');

TEST_FINISHED();
END_METHOD

METHOD PUBLIC Check_DWORD_TO_LINT_Min
VAR
	value : DWORD := DatatypeLimits.DWORD_MIN_VALUE;
	actual : LINT;
	converted : BOOL;
	equal : BOOL;
END_VAR
TEST('Check_DWORD_TO_LINT_Min');

// @TEST-RUN
converted := TryConvert_DWORD_TO_Destination(value, actual);
equal := actual = DWORD_TO_LINT(value);

// @TEST-ASSERT
AssertTrue(Condition := equal, Message := 'Did not convert DWORD to LINT correctly');
AssertTrue(Condition := converted, Message := 'Did not report DWORD to LINT conversion was successful');

TEST_FINISHED();
END_METHOD

METHOD PUBLIC Check_DWORD_TO_LINT_Max
VAR
	value : DWORD := DatatypeLimits.DWORD_MAX_VALUE;
	actual : LINT;
	converted : BOOL;
	equal : BOOL;
END_VAR
TEST('Check_DWORD_TO_LINT_Max');

// @TEST-RUN
converted := TryConvert_DWORD_TO_Destination(value, actual);
equal := actual = DWORD_TO_LINT(value);

// @TEST-ASSERT
AssertTrue(Condition := equal, Message := 'Did not convert DWORD to LINT correctly');
AssertTrue(Condition := converted, Message := 'Did not report DWORD to LINT conversion was successful');

TEST_FINISHED();
END_METHOD

METHOD PUBLIC Check_DWORD_TO_LREAL_Min
VAR
	value : DWORD := DatatypeLimits.DWORD_MIN_VALUE;
	actual : LREAL;
	converted : BOOL;
	equal : BOOL;
END_VAR
TEST('Check_DWORD_TO_LREAL_Min');

// @TEST-RUN
converted := TryConvert_DWORD_TO_Destination(value, actual);
equal := actual = DWORD_TO_LREAL(value);

// @TEST-ASSERT
AssertTrue(Condition := equal, Message := 'Did not convert DWORD to LREAL correctly');
AssertTrue(Condition := converted, Message := 'Did not report DWORD to LREAL conversion was successful');

TEST_FINISHED();
END_METHOD

METHOD PUBLIC Check_DWORD_TO_LREAL_Max
VAR
	value : DWORD := DatatypeLimits.DWORD_MAX_VALUE;
	actual : LREAL;
	converted : BOOL;
	equal : BOOL;
END_VAR
TEST('Check_DWORD_TO_LREAL_Max');

// @TEST-RUN
converted := TryConvert_DWORD_TO_Destination(value, actual);
equal := actual = DWORD_TO_LREAL(value);

// @TEST-ASSERT
AssertTrue(Condition := equal, Message := 'Did not convert DWORD to LREAL correctly');
AssertTrue(Condition := converted, Message := 'Did not report DWORD to LREAL conversion was successful');

TEST_FINISHED();
END_METHOD

METHOD PUBLIC Check_DWORD_TO_LWORD_Min
VAR
	value : DWORD := DatatypeLimits.DWORD_MIN_VALUE;
	actual : LWORD;
	converted : BOOL;
	equal : BOOL;
END_VAR
TEST('Check_DWORD_TO_LWORD_Min');

// @TEST-RUN
converted := TryConvert_DWORD_TO_Destination(value, actual);
equal := actual = DWORD_TO_LWORD(value);

// @TEST-ASSERT
AssertTrue(Condition := equal, Message := 'Did not convert DWORD to LWORD correctly');
AssertTrue(Condition := converted, Message := 'Did not report DWORD to LWORD conversion was successful');

TEST_FINISHED();
END_METHOD

METHOD PUBLIC Check_DWORD_TO_LWORD_Max
VAR
	value : DWORD := DatatypeLimits.DWORD_MAX_VALUE;
	actual : LWORD;
	converted : BOOL;
	equal : BOOL;
END_VAR
TEST('Check_DWORD_TO_LWORD_Max');

// @TEST-RUN
converted := TryConvert_DWORD_TO_Destination(value, actual);
equal := actual = DWORD_TO_LWORD(value);

// @TEST-ASSERT
AssertTrue(Condition := equal, Message := 'Did not convert DWORD to LWORD correctly');
AssertTrue(Condition := converted, Message := 'Did not report DWORD to LWORD conversion was successful');

TEST_FINISHED();
END_METHOD

METHOD PUBLIC Check_DWORD_TO_REAL_Min
VAR
	value : DWORD := DatatypeLimits.DWORD_MIN_VALUE;
	actual : REAL;
	converted : BOOL;
	equal : BOOL;
END_VAR
TEST('Check_DWORD_TO_REAL_Min');

// @TEST-RUN
converted := TryConvert_DWORD_TO_Destination(value, actual);
equal := actual = DWORD_TO_REAL(value);

// @TEST-ASSERT
AssertTrue(Condition := equal, Message := 'Did not convert DWORD to REAL correctly');
AssertTrue(Condition := converted, Message := 'Did not report DWORD to REAL conversion was successful');

TEST_FINISHED();
END_METHOD

METHOD PUBLIC Check_DWORD_TO_REAL_Max
VAR
	value : DWORD := DatatypeLimits.DWORD_MAX_VALUE;
	actual : REAL;
	converted : BOOL;
	equal : BOOL;
END_VAR
TEST('Check_DWORD_TO_REAL_Max');

// @TEST-RUN
converted := TryConvert_DWORD_TO_Destination(value, actual);
equal := actual = DWORD_TO_REAL(value);

// @TEST-ASSERT
AssertTrue(Condition := equal, Message := 'Did not convert DWORD to REAL correctly');
AssertTrue(Condition := converted, Message := 'Did not report DWORD to REAL conversion was successful');

TEST_FINISHED();
END_METHOD

METHOD PUBLIC Check_DWORD_TO_SINT_Min
VAR
	value : DWORD := DatatypeLimits.DWORD_MIN_VALUE;
	actual : SINT;
	converted : BOOL;
	equal : BOOL;
END_VAR
TEST('Check_DWORD_TO_SINT_Min');

// @TEST-RUN
converted := TryConvert_DWORD_TO_Destination(value, actual);
equal := actual = DWORD_TO_SINT(value);

// @TEST-ASSERT
AssertTrue(Condition := equal, Message := 'Did not convert DWORD to SINT correctly');
AssertTrue(Condition := converted, Message := 'Did not report DWORD to SINT conversion was successful');

TEST_FINISHED();
END_METHOD

METHOD PUBLIC Check_DWORD_TO_SINT_TooHigh
VAR
	value : DWORD := DatatypeLimits.DWORD_MAX_VALUE;
	actual : SINT;
	converted : BOOL;
END_VAR
TEST('Check_DWORD_TO_SINT_TooHigh');

// @TEST-RUN
converted := TryConvert_DWORD_TO_Destination(value, actual);

// @TEST-ASSERT
AssertFalse(Condition := converted, Message := 'Did not report DWORD to SINT conversion was prevented');

TEST_FINISHED();
END_METHOD

METHOD PUBLIC Check_DWORD_TO_SINT_Max
VAR
	value : DWORD := DatatypeLimits.MAX_VALUE_OF_DWORD_WHICH_CAN_BE_HELD_IN_A_SINT;
	actual : SINT;
	converted : BOOL;
	equal : BOOL;
END_VAR
TEST('Check_DWORD_TO_SINT_Max');

// @TEST-RUN
converted := TryConvert_DWORD_TO_Destination(value, actual);
equal := actual = DWORD_TO_SINT(value);

// @TEST-ASSERT
AssertTrue(Condition := equal, Message := 'Did not convert DWORD to SINT correctly');
AssertTrue(Condition := converted, Message := 'Did not report DWORD to SINT conversion was successful');

TEST_FINISHED();
END_METHOD

METHOD PUBLIC Check_DWORD_TO_STRING_Min
VAR
	value : DWORD := DatatypeLimits.DWORD_MIN_VALUE;
	actual : STRING;
	converted : BOOL;
	equal : BOOL;
END_VAR
TEST('Check_DWORD_TO_STRING_Min');

// @TEST-RUN
converted := TryConvert_DWORD_TO_Destination(value, actual);
equal := actual = DWORD_TO_STRING(value);

// @TEST-ASSERT
AssertTrue(Condition := equal, Message := 'Did not convert DWORD to STRING correctly');
AssertTrue(Condition := converted, Message := 'Did not report DWORD to STRING conversion was successful');

TEST_FINISHED();
END_METHOD

METHOD PUBLIC Check_DWORD_TO_STRING_Max
VAR
	value : DWORD := DatatypeLimits.DWORD_MAX_VALUE;
	actual : STRING;
	converted : BOOL;
	equal : BOOL;
END_VAR
TEST('Check_DWORD_TO_STRING_Max');

// @TEST-RUN
converted := TryConvert_DWORD_TO_Destination(value, actual);
equal := actual = DWORD_TO_STRING(value);

// @TEST-ASSERT
AssertTrue(Condition := equal, Message := 'Did not convert DWORD to STRING correctly');
AssertTrue(Condition := converted, Message := 'Did not report DWORD to STRING conversion was successful');

TEST_FINISHED();
END_METHOD

METHOD PUBLIC Check_DWORD_TO_TIME_Min
VAR
	value : DWORD := DatatypeLimits.DWORD_MIN_VALUE;
	actual : TIME;
	converted : BOOL;
	equal : BOOL;
END_VAR
TEST('Check_DWORD_TO_TIME_Min');

// @TEST-RUN
converted := TryConvert_DWORD_TO_Destination(value, actual);
equal := actual = DWORD_TO_TIME(value);

// @TEST-ASSERT
AssertTrue(Condition := equal, Message := 'Did not convert DWORD to TIME correctly');
AssertTrue(Condition := converted, Message := 'Did not report DWORD to TIME conversion was successful');

TEST_FINISHED();
END_METHOD

METHOD PUBLIC Check_DWORD_TO_TIME_Max
VAR
	value : DWORD := DatatypeLimits.DWORD_MAX_VALUE;
	actual : TIME;
	converted : BOOL;
	equal : BOOL;
END_VAR
TEST('Check_DWORD_TO_TIME_Max');

// @TEST-RUN
converted := TryConvert_DWORD_TO_Destination(value, actual);
equal := actual = DWORD_TO_TIME(value);

// @TEST-ASSERT
AssertTrue(Condition := equal, Message := 'Did not convert DWORD to TIME correctly');
AssertTrue(Condition := converted, Message := 'Did not report DWORD to TIME conversion was successful');

TEST_FINISHED();
END_METHOD

METHOD PUBLIC Check_DWORD_TO_TOD_Min
VAR
	value : DWORD := DatatypeLimits.DWORD_MIN_VALUE;
	actual : TOD;
	converted : BOOL;
	equal : BOOL;
END_VAR
TEST('Check_DWORD_TO_TOD_Min');

// @TEST-RUN
converted := TryConvert_DWORD_TO_Destination(value, actual);
equal := actual = DWORD_TO_TOD(value);

// @TEST-ASSERT
AssertTrue(Condition := equal, Message := 'Did not convert DWORD to TOD correctly');
AssertTrue(Condition := converted, Message := 'Did not report DWORD to TOD conversion was successful');

TEST_FINISHED();
END_METHOD

METHOD PUBLIC Check_DWORD_TO_TOD_TooHigh
VAR
	value : DWORD := DatatypeLimits.DWORD_MAX_VALUE;
	actual : TOD;
	converted : BOOL;
END_VAR
TEST('Check_DWORD_TO_TOD_TooHigh');

// @TEST-RUN
converted := TryConvert_DWORD_TO_Destination(value, actual);

// @TEST-ASSERT
AssertFalse(Condition := converted, Message := 'Did not report DWORD to TOD conversion was prevented');

TEST_FINISHED();
END_METHOD

METHOD PUBLIC Check_DWORD_TO_TOD_Max
VAR
	value : DWORD := DatatypeLimits.MAX_VALUE_OF_DWORD_WHICH_CAN_BE_HELD_IN_A_TOD;
	actual : TOD;
	converted : BOOL;
	equal : BOOL;
END_VAR
TEST('Check_DWORD_TO_TOD_Max');

// @TEST-RUN
converted := TryConvert_DWORD_TO_Destination(value, actual);
equal := actual = DWORD_TO_TOD(value);

// @TEST-ASSERT
AssertTrue(Condition := equal, Message := 'Did not convert DWORD to TOD correctly');
AssertTrue(Condition := converted, Message := 'Did not report DWORD to TOD conversion was successful');

TEST_FINISHED();
END_METHOD

METHOD PUBLIC Check_DWORD_TO_UDINT_Min
VAR
	value : DWORD := DatatypeLimits.DWORD_MIN_VALUE;
	actual : UDINT;
	converted : BOOL;
	equal : BOOL;
END_VAR
TEST('Check_DWORD_TO_UDINT_Min');

// @TEST-RUN
converted := TryConvert_DWORD_TO_Destination(value, actual);
equal := actual = DWORD_TO_UDINT(value);

// @TEST-ASSERT
AssertTrue(Condition := equal, Message := 'Did not convert DWORD to UDINT correctly');
AssertTrue(Condition := converted, Message := 'Did not report DWORD to UDINT conversion was successful');

TEST_FINISHED();
END_METHOD

METHOD PUBLIC Check_DWORD_TO_UDINT_Max
VAR
	value : DWORD := DatatypeLimits.DWORD_MAX_VALUE;
	actual : UDINT;
	converted : BOOL;
	equal : BOOL;
END_VAR
TEST('Check_DWORD_TO_UDINT_Max');

// @TEST-RUN
converted := TryConvert_DWORD_TO_Destination(value, actual);
equal := actual = DWORD_TO_UDINT(value);

// @TEST-ASSERT
AssertTrue(Condition := equal, Message := 'Did not convert DWORD to UDINT correctly');
AssertTrue(Condition := converted, Message := 'Did not report DWORD to UDINT conversion was successful');

TEST_FINISHED();
END_METHOD

METHOD PUBLIC Check_DWORD_TO_UINT_Min
VAR
	value : DWORD := DatatypeLimits.DWORD_MIN_VALUE;
	actual : UINT;
	converted : BOOL;
	equal : BOOL;
END_VAR
TEST('Check_DWORD_TO_UINT_Min');

// @TEST-RUN
converted := TryConvert_DWORD_TO_Destination(value, actual);
equal := actual = DWORD_TO_UINT(value);

// @TEST-ASSERT
AssertTrue(Condition := equal, Message := 'Did not convert DWORD to UINT correctly');
AssertTrue(Condition := converted, Message := 'Did not report DWORD to UINT conversion was successful');

TEST_FINISHED();
END_METHOD

METHOD PUBLIC Check_DWORD_TO_UINT_TooHigh
VAR
	value : DWORD := DatatypeLimits.DWORD_MAX_VALUE;
	actual : UINT;
	converted : BOOL;
END_VAR
TEST('Check_DWORD_TO_UINT_TooHigh');

// @TEST-RUN
converted := TryConvert_DWORD_TO_Destination(value, actual);

// @TEST-ASSERT
AssertFalse(Condition := converted, Message := 'Did not report DWORD to UINT conversion was prevented');

TEST_FINISHED();
END_METHOD

METHOD PUBLIC Check_DWORD_TO_UINT_Max
VAR
	value : DWORD := DatatypeLimits.MAX_VALUE_OF_DWORD_WHICH_CAN_BE_HELD_IN_A_UINT;
	actual : UINT;
	converted : BOOL;
	equal : BOOL;
END_VAR
TEST('Check_DWORD_TO_UINT_Max');

// @TEST-RUN
converted := TryConvert_DWORD_TO_Destination(value, actual);
equal := actual = DWORD_TO_UINT(value);

// @TEST-ASSERT
AssertTrue(Condition := equal, Message := 'Did not convert DWORD to UINT correctly');
AssertTrue(Condition := converted, Message := 'Did not report DWORD to UINT conversion was successful');

TEST_FINISHED();
END_METHOD

METHOD PUBLIC Check_DWORD_TO_ULINT_Min
VAR
	value : DWORD := DatatypeLimits.DWORD_MIN_VALUE;
	actual : ULINT;
	converted : BOOL;
	equal : BOOL;
END_VAR
TEST('Check_DWORD_TO_ULINT_Min');

// @TEST-RUN
converted := TryConvert_DWORD_TO_Destination(value, actual);
equal := actual = DWORD_TO_ULINT(value);

// @TEST-ASSERT
AssertTrue(Condition := equal, Message := 'Did not convert DWORD to ULINT correctly');
AssertTrue(Condition := converted, Message := 'Did not report DWORD to ULINT conversion was successful');

TEST_FINISHED();
END_METHOD

METHOD PUBLIC Check_DWORD_TO_ULINT_Max
VAR
	value : DWORD := DatatypeLimits.DWORD_MAX_VALUE;
	actual : ULINT;
	converted : BOOL;
	equal : BOOL;
END_VAR
TEST('Check_DWORD_TO_ULINT_Max');

// @TEST-RUN
converted := TryConvert_DWORD_TO_Destination(value, actual);
equal := actual = DWORD_TO_ULINT(value);

// @TEST-ASSERT
AssertTrue(Condition := equal, Message := 'Did not convert DWORD to ULINT correctly');
AssertTrue(Condition := converted, Message := 'Did not report DWORD to ULINT conversion was successful');

TEST_FINISHED();
END_METHOD

METHOD PUBLIC Check_DWORD_TO_USINT_Min
VAR
	value : DWORD := DatatypeLimits.DWORD_MIN_VALUE;
	actual : USINT;
	converted : BOOL;
	equal : BOOL;
END_VAR
TEST('Check_DWORD_TO_USINT_Min');

// @TEST-RUN
converted := TryConvert_DWORD_TO_Destination(value, actual);
equal := actual = DWORD_TO_USINT(value);

// @TEST-ASSERT
AssertTrue(Condition := equal, Message := 'Did not convert DWORD to USINT correctly');
AssertTrue(Condition := converted, Message := 'Did not report DWORD to USINT conversion was successful');

TEST_FINISHED();
END_METHOD

METHOD PUBLIC Check_DWORD_TO_USINT_TooHigh
VAR
	value : DWORD := DatatypeLimits.DWORD_MAX_VALUE;
	actual : USINT;
	converted : BOOL;
END_VAR
TEST('Check_DWORD_TO_USINT_TooHigh');

// @TEST-RUN
converted := TryConvert_DWORD_TO_Destination(value, actual);

// @TEST-ASSERT
AssertFalse(Condition := converted, Message := 'Did not report DWORD to USINT conversion was prevented');

TEST_FINISHED();
END_METHOD

METHOD PUBLIC Check_DWORD_TO_USINT_Max
VAR
	value : DWORD := DatatypeLimits.MAX_VALUE_OF_DWORD_WHICH_CAN_BE_HELD_IN_A_USINT;
	actual : USINT;
	converted : BOOL;
	equal : BOOL;
END_VAR
TEST('Check_DWORD_TO_USINT_Max');

// @TEST-RUN
converted := TryConvert_DWORD_TO_Destination(value, actual);
equal := actual = DWORD_TO_USINT(value);

// @TEST-ASSERT
AssertTrue(Condition := equal, Message := 'Did not convert DWORD to USINT correctly');
AssertTrue(Condition := converted, Message := 'Did not report DWORD to USINT conversion was successful');

TEST_FINISHED();
END_METHOD

METHOD PUBLIC Check_DWORD_TO_WORD_Min
VAR
	value : DWORD := DatatypeLimits.DWORD_MIN_VALUE;
	actual : WORD;
	converted : BOOL;
	equal : BOOL;
END_VAR
TEST('Check_DWORD_TO_WORD_Min');

// @TEST-RUN
converted := TryConvert_DWORD_TO_Destination(value, actual);
equal := actual = DWORD_TO_WORD(value);

// @TEST-ASSERT
AssertTrue(Condition := equal, Message := 'Did not convert DWORD to WORD correctly');
AssertTrue(Condition := converted, Message := 'Did not report DWORD to WORD conversion was successful');

TEST_FINISHED();
END_METHOD

METHOD PUBLIC Check_DWORD_TO_WORD_TooHigh
VAR
	value : DWORD := DatatypeLimits.DWORD_MAX_VALUE;
	actual : WORD;
	converted : BOOL;
END_VAR
TEST('Check_DWORD_TO_WORD_TooHigh');

// @TEST-RUN
converted := TryConvert_DWORD_TO_Destination(value, actual);

// @TEST-ASSERT
AssertFalse(Condition := converted, Message := 'Did not report DWORD to WORD conversion was prevented');

TEST_FINISHED();
END_METHOD

METHOD PUBLIC Check_DWORD_TO_WORD_Max
VAR
	value : DWORD := DatatypeLimits.MAX_VALUE_OF_DWORD_WHICH_CAN_BE_HELD_IN_A_WORD;
	actual : WORD;
	converted : BOOL;
	equal : BOOL;
END_VAR
TEST('Check_DWORD_TO_WORD_Max');

// @TEST-RUN
converted := TryConvert_DWORD_TO_Destination(value, actual);
equal := actual = DWORD_TO_WORD(value);

// @TEST-ASSERT
AssertTrue(Condition := equal, Message := 'Did not convert DWORD to WORD correctly');
AssertTrue(Condition := converted, Message := 'Did not report DWORD to WORD conversion was successful');

TEST_FINISHED();
END_METHOD

END_FUNCTION_BLOCK

// ---- Tests/LWORD_TO_TestSuite.TcPOU
FUNCTION_BLOCK PUBLIC LWORD_TO_TestSuite EXTENDS TcUnit.FB_TestSuite
VAR
END_VAR

Check_LWORD_TO_BOOL_Max();
Check_LWORD_TO_BOOL_Min();
Check_LWORD_TO_BYTE_Max();
Check_LWORD_TO_BYTE_Min();
Check_LWORD_TO_BYTE_TooHigh();
Check_LWORD_TO_WORD_Max();
Check_LWORD_TO_WORD_Min();
Check_LWORD_TO_WORD_TooHigh();
Check_LWORD_TO_DWORD_Max();
Check_LWORD_TO_DWORD_Min();
Check_LWORD_TO_DWORD_TooHigh();
Check_LWORD_TO_LWORD_Max();
Check_LWORD_TO_LWORD_Min();
Check_LWORD_TO_SINT_Max();
Check_LWORD_TO_SINT_Min();
Check_LWORD_TO_SINT_TooHigh();
Check_LWORD_TO_INT_Max();
Check_LWORD_TO_INT_Min();
Check_LWORD_TO_INT_TooHigh();
Check_LWORD_TO_DINT_Max();
Check_LWORD_TO_DINT_Min();
Check_LWORD_TO_DINT_TooHigh();
Check_LWORD_TO_LINT_Max();
Check_LWORD_TO_LINT_Min();
Check_LWORD_TO_LINT_TooHigh();
Check_LWORD_TO_USINT_Max();
Check_LWORD_TO_USINT_Min();
Check_LWORD_TO_USINT_TooHigh();
Check_LWORD_TO_UINT_Max();
Check_LWORD_TO_UINT_Min();
Check_LWORD_TO_UINT_TooHigh();
Check_LWORD_TO_UDINT_Max();
Check_LWORD_TO_UDINT_Min();
Check_LWORD_TO_UDINT_TooHigh();
Check_LWORD_TO_ULINT_Max();
Check_LWORD_TO_ULINT_Min();
Check_LWORD_TO_REAL_Max();
Check_LWORD_TO_REAL_Min();
Check_LWORD_TO_LREAL_Max();
Check_LWORD_TO_LREAL_Min();
Check_LWORD_TO_TIME_Max();
Check_LWORD_TO_TIME_Min();
Check_LWORD_TO_TIME_TooHigh();
Check_LWORD_TO_TOD_Max();
Check_LWORD_TO_TOD_Min();
Check_LWORD_TO_TOD_TooHigh();
Check_LWORD_TO_DATE_Max();
Check_LWORD_TO_DATE_Min();
Check_LWORD_TO_DATE_TooHigh();
Check_LWORD_TO_DT_Max();
Check_LWORD_TO_DT_Min();
Check_LWORD_TO_DT_TooHigh();
Check_LWORD_TO_STRING_Max();
Check_LWORD_TO_STRING_Min();

METHOD PUBLIC Check_LWORD_TO_BOOL_Min
VAR
	value : LWORD := DatatypeLimits.LWORD_MIN_VALUE;
	actual : BOOL;
	converted : BOOL;
	equal : BOOL;
END_VAR
TEST('Check_LWORD_TO_BOOL_Min');

// @TEST-RUN
converted := TryConvert_LWORD_TO_Destination(value, actual);
equal := actual = LWORD_TO_BOOL(value);

// @TEST-ASSERT
AssertTrue(Condition := equal, Message := 'Did not convert LWORD to BOOL correctly');
AssertTrue(Condition := converted, Message := 'Did not report LWORD to BOOL conversion was successful');

TEST_FINISHED();
END_METHOD

